END_VAR
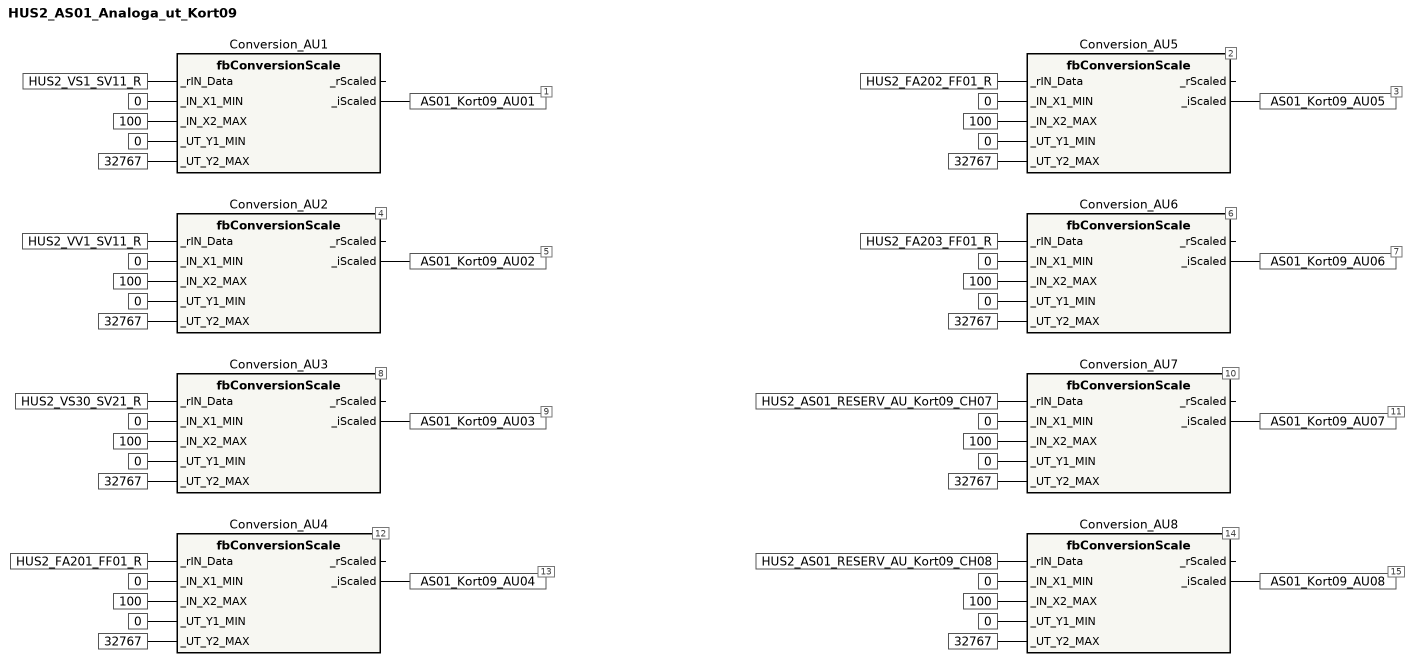
[picture p38: HUS2_AS01_Analoga_ut_Kort09 (CFC)]
_CFC_ (* Continuous Function Chart, elements in execution order *)
#0 Conversion_AU1:fbConversionScale(_rIN_Data: HUS2_VS1_SV11_R, _IN_X1_MIN: 0, _IN_X2_MAX: 100, _UT_Y1_MIN: 0, _UT_Y2_MAX: 32767)
#1 AS01_Kort09_AU01 <= #0._iScaled
#2 Conversion_AU5:fbConversionScale(_rIN_Data: HUS2_FA202_FF01_R, _IN_X1_MIN: 0, _IN_X2_MAX: 100, _UT_Y1_MIN: 0, _UT_Y2_MAX: 32767)
#3 AS01_Kort09_AU05 <= #2._iScaled
#4 Conversion_AU2:fbConversionScale(_rIN_Data: HUS2_VV1_SV11_R, _IN_X1_MIN: 0, _IN_X2_MAX: 100, _UT_Y1_MIN: 0, _UT_Y2_MAX: 32767)
#5 AS01_Kort09_AU02 <= #4._iScaled
#6 Conversion_AU6:fbConversionScale(_rIN_Data: HUS2_FA203_FF01_R, _IN_X1_MIN: 0, _IN_X2_MAX: 100, _UT_Y1_MIN: 0, _UT_Y2_MAX: 32767)
#7 AS01_Kort09_AU06 <= #6._iScaled
#8 Conversion_AU3:fbConversionScale(_rIN_Data: HUS2_VS30_SV21_R, _IN_X1_MIN: 0, _IN_X2_MAX: 100, _UT_Y1_MIN: 0, _UT_Y2_MAX: 32767)
#9 AS01_Kort09_AU03 <= #8._iScaled
#10 Conversion_AU7:fbConversionScale(_rIN_Data: HUS2_AS01_RESERV_AU_Kort09_CH07, _IN_X1_MIN: 0, _IN_X2_MAX: 100, _UT_Y1_MIN: 0, _UT_Y2_MAX: 32767)
#11 AS01_Kort09_AU07 <= #10._iScaled
#12 Conversion_AU4:fbConversionScale(_rIN_Data: HUS2_FA201_FF01_R, _IN_X1_MIN: 0, _IN_X2_MAX: 100, _UT_Y1_MIN: 0, _UT_Y2_MAX: 32767)
#13 AS01_Kort09_AU04 <= #12._iScaled
#14 Conversion_AU8:fbConversionScale(_rIN_Data: HUS2_AS01_RESERV_AU_Kort09_CH08, _IN_X1_MIN: 0, _IN_X2_MAX: 100, _UT_Y1_MIN: 0, _UT_Y2_MAX: 32767)
#15 AS01_Kort09_AU08 <= #14._iScaled
_END_CFC_
(* the same logic as Structured Text *)
Conversion_AU1(_rIN_Data := HUS2_VS1_SV11_R, _IN_X1_MIN := 0, _IN_X2_MAX := 100, _UT_Y1_MIN := 0, _UT_Y2_MAX := 32767);
AS01_Kort09_AU01 := Conversion_AU1._iScaled;
Conversion_AU5(_rIN_Data := HUS2_FA202_FF01_R, _IN_X1_MIN := 0, _IN_X2_MAX := 100, _UT_Y1_MIN := 0, _UT_Y2_MAX := 32767);
AS01_Kort09_AU05 := Conversion_AU5._iScaled;
Conversion_AU2(_rIN_Data := HUS2_VV1_SV11_R, _IN_X1_MIN := 0, _IN_X2_MAX := 100, _UT_Y1_MIN := 0, _UT_Y2_MAX := 32767);
AS01_Kort09_AU02 := Conversion_AU2._iScaled;
Conversion_AU6(_rIN_Data := HUS2_FA203_FF01_R, _IN_X1_MIN := 0, _IN_X2_MAX := 100, _UT_Y1_MIN := 0, _UT_Y2_MAX := 32767);
AS01_Kort09_AU06 := Conversion_AU6._iScaled;
Conversion_AU3(_rIN_Data := HUS2_VS30_SV21_R, _IN_X1_MIN := 0, _IN_X2_MAX := 100, _UT_Y1_MIN := 0, _UT_Y2_MAX := 32767);
AS01_Kort09_AU03 := Conversion_AU3._iScaled;
Conversion_AU7(_rIN_Data := HUS2_AS01_RESERV_AU_Kort09_CH07, _IN_X1_MIN := 0, _IN_X2_MAX := 100, _UT_Y1_MIN := 0, _UT_Y2_MAX := 32767);
AS01_Kort09_AU07 := Conversion_AU7._iScaled;
Conversion_AU4(_rIN_Data := HUS2_FA201_FF01_R, _IN_X1_MIN := 0, _IN_X2_MAX := 100, _UT_Y1_MIN := 0, _UT_Y2_MAX := 32767);
AS01_Kort09_AU04 := Conversion_AU4._iScaled;
Conversion_AU8(_rIN_Data := HUS2_AS01_RESERV_AU_Kort09_CH08, _IN_X1_MIN := 0, _IN_X2_MAX := 100, _UT_Y1_MIN := 0, _UT_Y2_MAX := 32767);
AS01_Kort09_AU08 := Conversion_AU8._iScaled;
END_PROGRAM

(* POU _IOs_Uppdelat_per_skåp/HUS2_AL01/_IO/HUS2_AL01_IO_MAIN, CFC *)
PROGRAM HUS2_AL01_IO_MAIN
VAR
END_VAR
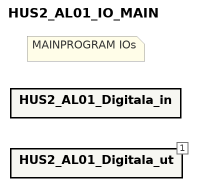
_CFC_ (* Continuous Function Chart, elements in execution order *)
(* MAINPROGRAM IOs *)
#0 HUS2_AL01_Digitala_in()
#1 HUS2_AL01_Digitala_ut()
_END_CFC_
(* the same logic as Structured Text *)
(* MAINPROGRAM IOs *)
HUS2_AL01_Digitala_in();
HUS2_AL01_Digitala_ut();
END_PROGRAM

(* POU _IOs_Uppdelat_per_skåp/HUS2_AL01/_IO/HUS2_AL01_Digitala_in, CFC *)
PROGRAM HUS2_AL01_Digitala_in

VAR


END_VAR
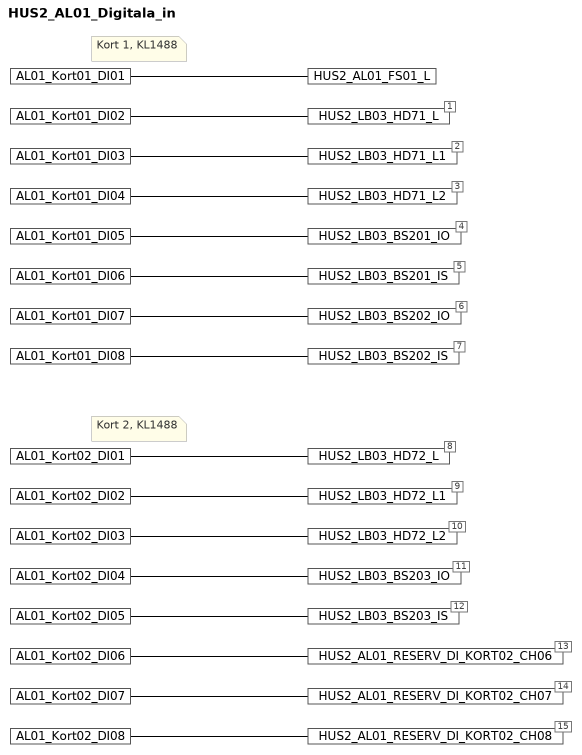
_CFC_ (* Continuous Function Chart, elements in execution order *)
(* Kort 1, KL1488 *)
(* Kort 2, KL1488 *)
#0 HUS2_AL01_FS01_L <= AL01_Kort01_DI01
#1 HUS2_LB03_HD71_L <= AL01_Kort01_DI02
#2 HUS2_LB03_HD71_L1 <= AL01_Kort01_DI03
#3 HUS2_LB03_HD71_L2 <= AL01_Kort01_DI04
#4 HUS2_LB03_BS201_IO <= AL01_Kort01_DI05
#5 HUS2_LB03_BS201_IS <= AL01_Kort01_DI06
#6 HUS2_LB03_BS202_IO <= AL01_Kort01_DI07
#7 HUS2_LB03_BS202_IS <= AL01_Kort01_DI08
#8 HUS2_LB03_HD72_L <= AL01_Kort02_DI01
#9 HUS2_LB03_HD72_L1 <= AL01_Kort02_DI02
#10 HUS2_LB03_HD72_L2 <= AL01_Kort02_DI03
#11 HUS2_LB03_BS203_IO <= AL01_Kort02_DI04
#12 HUS2_LB03_BS203_IS <= AL01_Kort02_DI05
#13 HUS2_AL01_RESERV_DI_KORT02_CH06 <= AL01_Kort02_DI06
#14 HUS2_AL01_RESERV_DI_KORT02_CH07 <= AL01_Kort02_DI07
#15 HUS2_AL01_RESERV_DI_KORT02_CH08 <= AL01_Kort02_DI08
_END_CFC_
(* the same logic as Structured Text *)
(* Kort 1, KL1488 *)
(* Kort 2, KL1488 *)
HUS2_AL01_FS01_L := AL01_Kort01_DI01;
HUS2_LB03_HD71_L := AL01_Kort01_DI02;
HUS2_LB03_HD71_L1 := AL01_Kort01_DI03;
HUS2_LB03_HD71_L2 := AL01_Kort01_DI04;
HUS2_LB03_BS201_IO := AL01_Kort01_DI05;
HUS2_LB03_BS201_IS := AL01_Kort01_DI06;
HUS2_LB03_BS202_IO := AL01_Kort01_DI07;
HUS2_LB03_BS202_IS := AL01_Kort01_DI08;
HUS2_LB03_HD72_L := AL01_Kort02_DI01;
HUS2_LB03_HD72_L1 := AL01_Kort02_DI02;
HUS2_LB03_HD72_L2 := AL01_Kort02_DI03;
HUS2_LB03_BS203_IO := AL01_Kort02_DI04;
HUS2_LB03_BS203_IS := AL01_Kort02_DI05;
HUS2_AL01_RESERV_DI_KORT02_CH06 := AL01_Kort02_DI06;
HUS2_AL01_RESERV_DI_KORT02_CH07 := AL01_Kort02_DI07;
HUS2_AL01_RESERV_DI_KORT02_CH08 := AL01_Kort02_DI08;
END_PROGRAM

(* POU _IOs_Uppdelat_per_skåp/HUS2_AL01/_IO/HUS2_AL01_Digitala_ut, CFC *)
PROGRAM HUS2_AL01_Digitala_ut


VAR
END_VAR
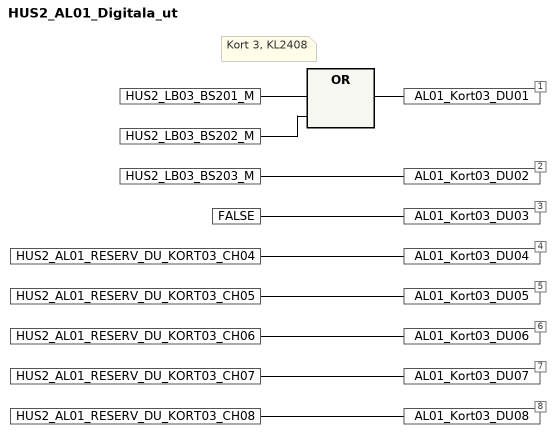
_CFC_ (* Continuous Function Chart, elements in execution order *)
(* Kort 3, KL2408 *)
#0 OR(HUS2_LB03_BS201_M, HUS2_LB03_BS202_M)
#1 AL01_Kort03_DU01 <= #0
#2 AL01_Kort03_DU02 <= HUS2_LB03_BS203_M
#3 AL01_Kort03_DU03 <= FALSE
#4 AL01_Kort03_DU04 <= HUS2_AL01_RESERV_DU_KORT03_CH04
#5 AL01_Kort03_DU05 <= HUS2_AL01_RESERV_DU_KORT03_CH05
#6 AL01_Kort03_DU06 <= HUS2_AL01_RESERV_DU_KORT03_CH06
#7 AL01_Kort03_DU07 <= HUS2_AL01_RESERV_DU_KORT03_CH07
#8 AL01_Kort03_DU08 <= HUS2_AL01_RESERV_DU_KORT03_CH08
_END_CFC_
(* the same logic as Structured Text *)
(* Kort 3, KL2408 *)
AL01_Kort03_DU01 := HUS2_LB03_BS201_M OR HUS2_LB03_BS202_M;
AL01_Kort03_DU02 := HUS2_LB03_BS203_M;
AL01_Kort03_DU03 := FALSE;
AL01_Kort03_DU04 := HUS2_AL01_RESERV_DU_KORT03_CH04;
AL01_Kort03_DU05 := HUS2_AL01_RESERV_DU_KORT03_CH05;
AL01_Kort03_DU06 := HUS2_AL01_RESERV_DU_KORT03_CH06;
AL01_Kort03_DU07 := HUS2_AL01_RESERV_DU_KORT03_CH07;
AL01_Kort03_DU08 := HUS2_AL01_RESERV_DU_KORT03_CH08;
END_PROGRAM

(* POU _IOs_Uppdelat_per_skåp/HUS3_AS03/_IO/HUS3_AS03_IO_MAIN, CFC *)
PROGRAM HUS3_AS03_IO_MAIN
VAR
END_VAR
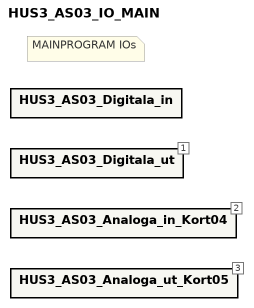
_CFC_ (* Continuous Function Chart, elements in execution order *)
(* MAINPROGRAM IOs *)
#0 HUS3_AS03_Digitala_in()
#1 HUS3_AS03_Digitala_ut()
#2 HUS3_AS03_Analoga_in_Kort04()
#3 HUS3_AS03_Analoga_ut_Kort05()
_END_CFC_
(* the same logic as Structured Text *)
(* MAINPROGRAM IOs *)
HUS3_AS03_Digitala_in();
HUS3_AS03_Digitala_ut();
HUS3_AS03_Analoga_in_Kort04();
HUS3_AS03_Analoga_ut_Kort05();
END_PROGRAM

(* POU _IOs_Uppdelat_per_skåp/HUS3_AS03/_IO/HUS3_AS03_Digitala_in, CFC *)
PROGRAM HUS3_AS03_Digitala_in

VAR


END_VAR
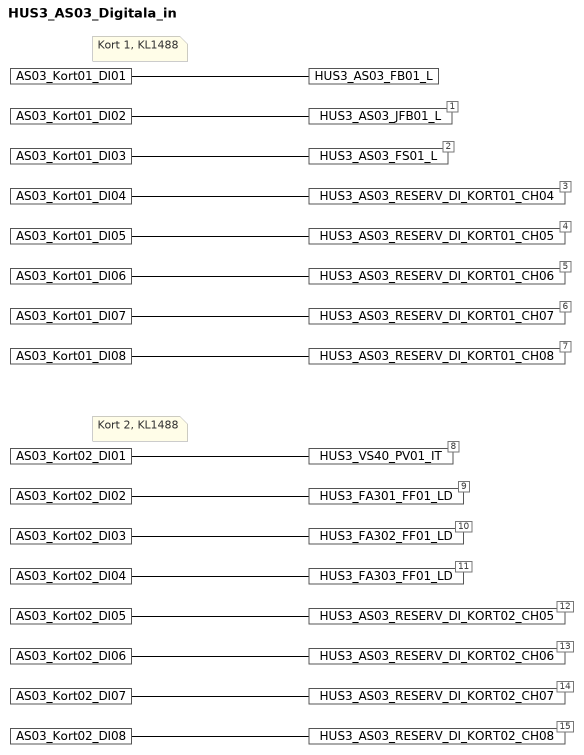
_CFC_ (* Continuous Function Chart, elements in execution order *)
(* Kort 2, KL1488 *)
(* Kort 1, KL1488 *)
#0 HUS3_AS03_FB01_L <= AS03_Kort01_DI01
#1 HUS3_AS03_JFB01_L <= AS03_Kort01_DI02
#2 HUS3_AS03_FS01_L <= AS03_Kort01_DI03
#3 HUS3_AS03_RESERV_DI_KORT01_CH04 <= AS03_Kort01_DI04
#4 HUS3_AS03_RESERV_DI_KORT01_CH05 <= AS03_Kort01_DI05
#5 HUS3_AS03_RESERV_DI_KORT01_CH06 <= AS03_Kort01_DI06
#6 HUS3_AS03_RESERV_DI_KORT01_CH07 <= AS03_Kort01_DI07
#7 HUS3_AS03_RESERV_DI_KORT01_CH08 <= AS03_Kort01_DI08
#8 HUS3_VS40_PV01_IT <= AS03_Kort02_DI01
#9 HUS3_FA301_FF01_LD <= AS03_Kort02_DI02
#10 HUS3_FA302_FF01_LD <= AS03_Kort02_DI03
#11 HUS3_FA303_FF01_LD <= AS03_Kort02_DI04
#12 HUS3_AS03_RESERV_DI_KORT02_CH05 <= AS03_Kort02_DI05
#13 HUS3_AS03_RESERV_DI_KORT02_CH06 <= AS03_Kort02_DI06
#14 HUS3_AS03_RESERV_DI_KORT02_CH07 <= AS03_Kort02_DI07
#15 HUS3_AS03_RESERV_DI_KORT02_CH08 <= AS03_Kort02_DI08
_END_CFC_
(* the same logic as Structured Text *)
(* Kort 2, KL1488 *)
(* Kort 1, KL1488 *)
HUS3_AS03_FB01_L := AS03_Kort01_DI01;
HUS3_AS03_JFB01_L := AS03_Kort01_DI02;
HUS3_AS03_FS01_L := AS03_Kort01_DI03;
HUS3_AS03_RESERV_DI_KORT01_CH04 := AS03_Kort01_DI04;
HUS3_AS03_RESERV_DI_KORT01_CH05 := AS03_Kort01_DI05;
HUS3_AS03_RESERV_DI_KORT01_CH06 := AS03_Kort01_DI06;
HUS3_AS03_RESERV_DI_KORT01_CH07 := AS03_Kort01_DI07;
HUS3_AS03_RESERV_DI_KORT01_CH08 := AS03_Kort01_DI08;
HUS3_VS40_PV01_IT := AS03_Kort02_DI01;
HUS3_FA301_FF01_LD := AS03_Kort02_DI02;
HUS3_FA302_FF01_LD := AS03_Kort02_DI03;
HUS3_FA303_FF01_LD := AS03_Kort02_DI04;
HUS3_AS03_RESERV_DI_KORT02_CH05 := AS03_Kort02_DI05;
HUS3_AS03_RESERV_DI_KORT02_CH06 := AS03_Kort02_DI06;
HUS3_AS03_RESERV_DI_KORT02_CH07 := AS03_Kort02_DI07;
HUS3_AS03_RESERV_DI_KORT02_CH08 := AS03_Kort02_DI08;
END_PROGRAM

(* POU _IOs_Uppdelat_per_skåp/HUS3_AS03/_IO/HUS3_AS03_Digitala_ut, CFC *)
PROGRAM HUS3_AS03_Digitala_ut


VAR

END_VAR
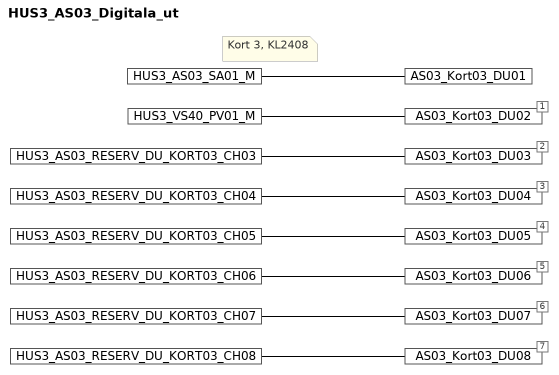
_CFC_ (* Continuous Function Chart, elements in execution order *)
(* Kort 3, KL2408 *)
#0 AS03_Kort03_DU01 <= HUS3_AS03_SA01_M
#1 AS03_Kort03_DU02 <= HUS3_VS40_PV01_M
#2 AS03_Kort03_DU03 <= HUS3_AS03_RESERV_DU_KORT03_CH03
#3 AS03_Kort03_DU04 <= HUS3_AS03_RESERV_DU_KORT03_CH04
#4 AS03_Kort03_DU05 <= HUS3_AS03_RESERV_DU_KORT03_CH05
#5 AS03_Kort03_DU06 <= HUS3_AS03_RESERV_DU_KORT03_CH06
#6 AS03_Kort03_DU07 <= HUS3_AS03_RESERV_DU_KORT03_CH07
#7 AS03_Kort03_DU08 <= HUS3_AS03_RESERV_DU_KORT03_CH08
_END_CFC_
(* the same logic as Structured Text *)
(* Kort 3, KL2408 *)
AS03_Kort03_DU01 := HUS3_AS03_SA01_M;
AS03_Kort03_DU02 := HUS3_VS40_PV01_M;
AS03_Kort03_DU03 := HUS3_AS03_RESERV_DU_KORT03_CH03;
AS03_Kort03_DU04 := HUS3_AS03_RESERV_DU_KORT03_CH04;
AS03_Kort03_DU05 := HUS3_AS03_RESERV_DU_KORT03_CH05;
AS03_Kort03_DU06 := HUS3_AS03_RESERV_DU_KORT03_CH06;
AS03_Kort03_DU07 := HUS3_AS03_RESERV_DU_KORT03_CH07;
AS03_Kort03_DU08 := HUS3_AS03_RESERV_DU_KORT03_CH08;
END_PROGRAM

(* POU _IOs_Uppdelat_per_skåp/HUS3_AS03/_IO/ANALOGA IN/Kort04/HUS3_AS03_Analoga_in_Kort04, CFC *)
PROGRAM HUS3_AS03_Analoga_in_Kort04
VAR
	bLG01: BOOL;
	bLG02: BOOL;
	bLG03: BOOL;
	bLG04: BOOL;
	bLG05: BOOL;
	bLG06: BOOL;
	bLG07: BOOL;
	bLG08: BOOL;

(*TEMP*)
	FT1:INT;
	LG_FL1:INT;
	FT2:INT;
	LG_FL2:INT;
	FT3:INT;
	LG_FL3:INT;
	FT4:INT;
	LG_FL4:INT;
	FT5:INT;
	LG_FL5:INT;
	FT6:INT;
	LG_FL6:INT;
	FT7:INT;
	LG_FL7:INT;
	FT8:INT;
	LG_FL8:INT;

END_VAR
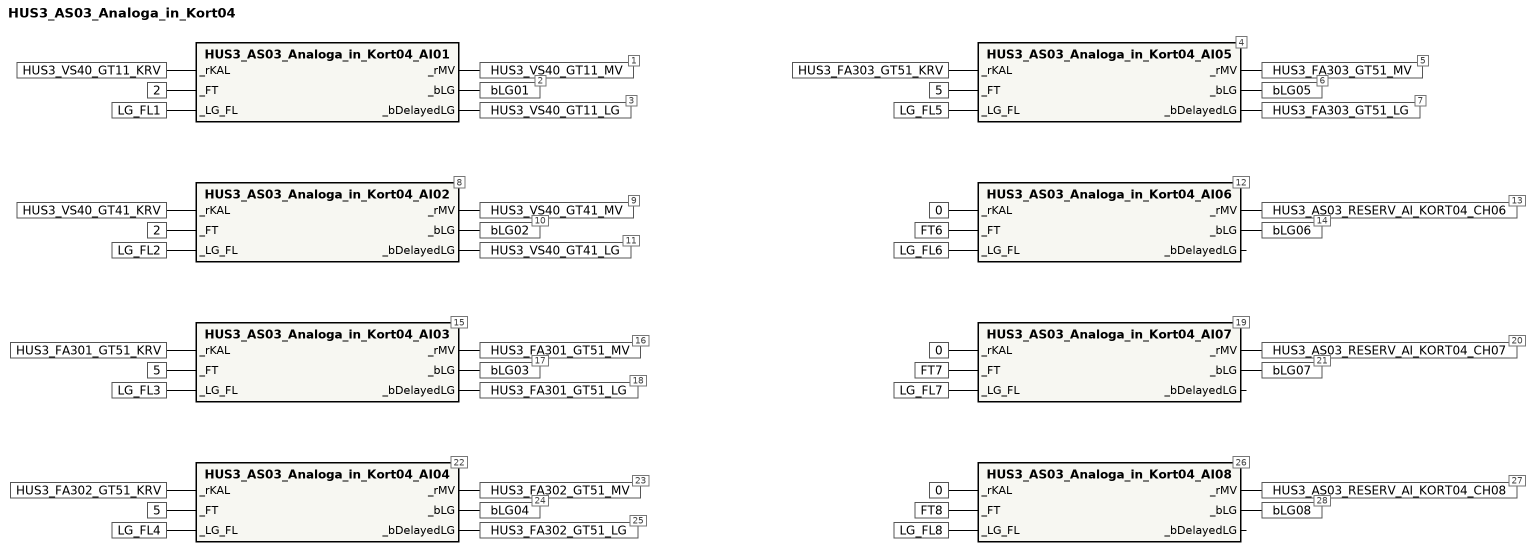
_CFC_ (* Continuous Function Chart, elements in execution order *)
#0 HUS3_AS03_Analoga_in_Kort04_AI01(_rKAL: HUS3_VS40_GT11_KRV, _FT: 2, _LG_FL: LG_FL1)
#1 HUS3_VS40_GT11_MV <= #0._rMV
#2 bLG01 <= #0._bLG
#3 HUS3_VS40_GT11_LG <= #0._bDelayedLG
#4 HUS3_AS03_Analoga_in_Kort04_AI05(_rKAL: HUS3_FA303_GT51_KRV, _FT: 5, _LG_FL: LG_FL5)
#5 HUS3_FA303_GT51_MV <= #4._rMV
#6 bLG05 <= #4._bLG
#7 HUS3_FA303_GT51_LG <= #4._bDelayedLG
#8 HUS3_AS03_Analoga_in_Kort04_AI02(_rKAL: HUS3_VS40_GT41_KRV, _FT: 2, _LG_FL: LG_FL2)
#9 HUS3_VS40_GT41_MV <= #8._rMV
#10 bLG02 <= #8._bLG
#11 HUS3_VS40_GT41_LG <= #8._bDelayedLG
#12 HUS3_AS03_Analoga_in_Kort04_AI06(_rKAL: 0, _FT: FT6, _LG_FL: LG_FL6)
#13 HUS3_AS03_RESERV_AI_KORT04_CH06 <= #12._rMV
#14 bLG06 <= #12._bLG
#15 HUS3_AS03_Analoga_in_Kort04_AI03(_rKAL: HUS3_FA301_GT51_KRV, _FT: 5, _LG_FL: LG_FL3)
#16 HUS3_FA301_GT51_MV <= #15._rMV
#17 bLG03 <= #15._bLG
#18 HUS3_FA301_GT51_LG <= #15._bDelayedLG
#19 HUS3_AS03_Analoga_in_Kort04_AI07(_rKAL: 0, _FT: FT7, _LG_FL: LG_FL7)
#20 HUS3_AS03_RESERV_AI_KORT04_CH07 <= #19._rMV
#21 bLG07 <= #19._bLG
#22 HUS3_AS03_Analoga_in_Kort04_AI04(_rKAL: HUS3_FA302_GT51_KRV, _FT: 5, _LG_FL: LG_FL4)
#23 HUS3_FA302_GT51_MV <= #22._rMV
#24 bLG04 <= #22._bLG
#25 HUS3_FA302_GT51_LG <= #22._bDelayedLG
#26 HUS3_AS03_Analoga_in_Kort04_AI08(_rKAL: 0, _FT: FT8, _LG_FL: LG_FL8)
#27 HUS3_AS03_RESERV_AI_KORT04_CH08 <= #26._rMV
#28 bLG08 <= #26._bLG
_END_CFC_
(* the same logic as Structured Text *)
HUS3_AS03_Analoga_in_Kort04_AI01(_rKAL := HUS3_VS40_GT11_KRV, _FT := 2, _LG_FL := LG_FL1);
HUS3_VS40_GT11_MV := HUS3_AS03_Analoga_in_Kort04_AI01._rMV;
bLG01 := HUS3_AS03_Analoga_in_Kort04_AI01._bLG;
HUS3_VS40_GT11_LG := HUS3_AS03_Analoga_in_Kort04_AI01._bDelayedLG;
HUS3_AS03_Analoga_in_Kort04_AI05(_rKAL := HUS3_FA303_GT51_KRV, _FT := 5, _LG_FL := LG_FL5);
HUS3_FA303_GT51_MV := HUS3_AS03_Analoga_in_Kort04_AI05._rMV;
bLG05 := HUS3_AS03_Analoga_in_Kort04_AI05._bLG;
HUS3_FA303_GT51_LG := HUS3_AS03_Analoga_in_Kort04_AI05._bDelayedLG;
HUS3_AS03_Analoga_in_Kort04_AI02(_rKAL := HUS3_VS40_GT41_KRV, _FT := 2, _LG_FL := LG_FL2);
HUS3_VS40_GT41_MV := HUS3_AS03_Analoga_in_Kort04_AI02._rMV;
bLG02 := HUS3_AS03_Analoga_in_Kort04_AI02._bLG;
HUS3_VS40_GT41_LG := HUS3_AS03_Analoga_in_Kort04_AI02._bDelayedLG;
HUS3_AS03_Analoga_in_Kort04_AI06(_rKAL := 0, _FT := FT6, _LG_FL := LG_FL6);
HUS3_AS03_RESERV_AI_KORT04_CH06 := HUS3_AS03_Analoga_in_Kort04_AI06._rMV;
bLG06 := HUS3_AS03_Analoga_in_Kort04_AI06._bLG;
HUS3_AS03_Analoga_in_Kort04_AI03(_rKAL := HUS3_FA301_GT51_KRV, _FT := 5, _LG_FL := LG_FL3);
HUS3_FA301_GT51_MV := HUS3_AS03_Analoga_in_Kort04_AI03._rMV;
bLG03 := HUS3_AS03_Analoga_in_Kort04_AI03._bLG;
HUS3_FA301_GT51_LG := HUS3_AS03_Analoga_in_Kort04_AI03._bDelayedLG;
HUS3_AS03_Analoga_in_Kort04_AI07(_rKAL := 0, _FT := FT7, _LG_FL := LG_FL7);
HUS3_AS03_RESERV_AI_KORT04_CH07 := HUS3_AS03_Analoga_in_Kort04_AI07._rMV;
bLG07 := HUS3_AS03_Analoga_in_Kort04_AI07._bLG;
HUS3_AS03_Analoga_in_Kort04_AI04(_rKAL := HUS3_FA302_GT51_KRV, _FT := 5, _LG_FL := LG_FL4);
HUS3_FA302_GT51_MV := HUS3_AS03_Analoga_in_Kort04_AI04._rMV;
bLG04 := HUS3_AS03_Analoga_in_Kort04_AI04._bLG;
HUS3_FA302_GT51_LG := HUS3_AS03_Analoga_in_Kort04_AI04._bDelayedLG;
HUS3_AS03_Analoga_in_Kort04_AI08(_rKAL := 0, _FT := FT8, _LG_FL := LG_FL8);
HUS3_AS03_RESERV_AI_KORT04_CH08 := HUS3_AS03_Analoga_in_Kort04_AI08._rMV;
bLG08 := HUS3_AS03_Analoga_in_Kort04_AI08._bLG;
END_PROGRAM

(* POU _IOs_Uppdelat_per_skåp/HUS3_AS03/_IO/ANALOGA IN/Kort04/HUS3_AS03_Analoga_in_Kort04_AI01, FAI *)
PROGRAM HUS3_AS03_Analoga_in_Kort04_AI01
(*#####################################   Temperature Sensor Ex2   ################################################################*)
VAR
	(*===========================Configuration of terminal==========================================*)
	fbConfigureKL32xx					:FB_HVACConfigureKL32xx;
	_byCtrlKL32xx                         			AT %Q*: BYTE;
	_iDataOutKL32xx                       		AT %Q*: INT;
	_iDataInKL32xx 					AT%I*:INT;(* Raw Value from the Terminal *)
	_byStatusKL32xx 			AT%I*:BYTE;(* Statusbyte from Terminal *)

	_bScanSensor              					: BOOL;
	_tTimeOut                 					: TIME := T#5s;
	_bSetSensor               					: BOOL;
	bReady                               				: BOOL;
	byOutStatus                          			: BYTE;
	iOutDataIn                           				: INT;
	_eBusTerminalKL32xx                   		: E_HVACBusTerminal_KL32xx;
	_eStatusScanSensorType                	: E_HVACSensorType;
	_bErrorGeneral                        			: BOOL;
	_byError                              				: BYTE;
	_bErrorCommunication                  		: BOOL;
	_bErrorBusTerminalNotSupported   	: BOOL;
	_bErrorSensorType                     		: BOOL;
	_bErrorScanSensor                     		: BOOL;
	(*========================================================================================*)

	_bReset_Local					:BOOL;
	_bSetDefaultTempSens			:BOOL;

	(*========================================================================================*)
	FBHVACTemperatureSensor: FB_HVACTemperatureSensor;
	eDataSecurityType					: E_HVACDataSecurityType:=1;
	bSetDefault								:BOOL;
	iRawValue								:INT;
	byStatusRawValue						:BYTE;
	bEnableLimitCtrl							:BOOL;
	bReset									:BOOL;
	bErrorGeneral					:BOOL;
	byError							:BYTE;
	bErrorShortCircuit				:BOOL;
	bErrorBrokenSensor				:BOOL;
	bErrorHighLimit					:BOOL;
	bErrorLowLimit					:BOOL;
	bErrorCycleTime					:BOOL;
	bInvalidParameter				:BOOL;
	rOffset									:REAL;
	rHighLimit								:REAL;
	rLowLimit								:REAL;
	rReplacementValue						:REAL;
	tFilterTime								:TIME;
	eTemperatureSensorMode				:E_HVACTemperatureSensorMode:=2;
	fbAlarmD: fbDelayedAlarmMinutes;

END_VAR

VAR_INPUT
	_rKAL						: REAL;	(*Kalibrering*)
	_FT						:INT;		(*Filtertid*)
	_LG_FL					:INT;		(* Larmfördröjning givarfel *)
END_VAR

VAR_OUTPUT
	_rMV						:REAL;		(* Mätvärde *)
	_bLG						:BOOL; 	(*Givarfel*)
	_bDelayedLG				:BOOL;	(* Fördröjt givarfel *)
END_VAR
(* body not read: cfc101 *)
END_PROGRAM

(* POU _IOs_Uppdelat_per_skåp/HUS3_AS03/_IO/ANALOGA IN/Kort04/HUS3_AS03_Analoga_in_Kort04_AI05, FAI *)
PROGRAM HUS3_AS03_Analoga_in_Kort04_AI05
(*#####################################   Temperature Sensor Ex2   ################################################################*)
VAR
	(*===========================Configuration of terminal==========================================*)
	fbConfigureKL32xx					:FB_HVACConfigureKL32xx;
	_byCtrlKL32xx                         			AT %Q*: BYTE;
	_iDataOutKL32xx                       		AT %Q*: INT;
	_iDataInKL32xx 					AT%I*:INT;(* Raw Value from the Terminal *)
	_byStatusKL32xx 			AT%I*:BYTE;(* Statusbyte from Terminal *)

	_bScanSensor              					: BOOL;
	_tTimeOut                 					: TIME := T#5s;
	_bSetSensor               					: BOOL;
	bReady                               				: BOOL;
	byOutStatus                          			: BYTE;
	iOutDataIn                           				: INT;
	_eBusTerminalKL32xx                   		: E_HVACBusTerminal_KL32xx;
	_eStatusScanSensorType                	: E_HVACSensorType;
	_bErrorGeneral                        			: BOOL;
	_byError                              				: BYTE;
	_bErrorCommunication                  		: BOOL;
	_bErrorBusTerminalNotSupported   	: BOOL;
	_bErrorSensorType                     		: BOOL;
	_bErrorScanSensor                     		: BOOL;
	(*========================================================================================*)

	_bReset_Local					:BOOL;
	_bSetDefaultTempSens			:BOOL;

	(*========================================================================================*)
	FBHVACTemperatureSensor: FB_HVACTemperatureSensor;
	eDataSecurityType					: E_HVACDataSecurityType:=1;
	bSetDefault								:BOOL;
	iRawValue								:INT;
	byStatusRawValue						:BYTE;
	bEnableLimitCtrl							:BOOL;
	bReset									:BOOL;
	bErrorGeneral					:BOOL;
	byError							:BYTE;
	bErrorShortCircuit				:BOOL;
	bErrorBrokenSensor				:BOOL;
	bErrorHighLimit					:BOOL;
	bErrorLowLimit					:BOOL;
	bErrorCycleTime					:BOOL;
	bInvalidParameter				:BOOL;
	rOffset									:REAL;
	rHighLimit								:REAL;
	rLowLimit								:REAL;
	rReplacementValue						:REAL;
	tFilterTime								:TIME;
	eTemperatureSensorMode				:E_HVACTemperatureSensorMode:=2;
	fbAlarmD: fbDelayedAlarmMinutes;

END_VAR

VAR_INPUT
	_rKAL						: REAL;	(*Kalibrering*)
	_FT						:INT;		(*Filtertid*)
	_LG_FL					:INT;		(* Larmfördröjning givarfel *)
END_VAR

VAR_OUTPUT
	_rMV						:REAL;		(* Mätvärde *)
	_bLG						:BOOL; 	(*Givarfel*)
	_bDelayedLG				:BOOL;	(* Fördröjt givarfel *)
END_VAR
(* body not read: cfc101 *)
END_PROGRAM

(* POU _IOs_Uppdelat_per_skåp/HUS3_AS03/_IO/ANALOGA IN/Kort04/HUS3_AS03_Analoga_in_Kort04_AI02, FAI *)
PROGRAM HUS3_AS03_Analoga_in_Kort04_AI02
(*#####################################   Temperature Sensor Ex2   ################################################################*)
VAR
	(*===========================Configuration of terminal==========================================*)
	fbConfigureKL32xx					:FB_HVACConfigureKL32xx;
	_byCtrlKL32xx                         			AT %Q*: BYTE;
	_iDataOutKL32xx                       		AT %Q*: INT;
	_iDataInKL32xx 					AT%I*:INT;(* Raw Value from the Terminal *)
	_byStatusKL32xx 			AT%I*:BYTE;(* Statusbyte from Terminal *)

	_bScanSensor              					: BOOL;
	_tTimeOut                 					: TIME := T#5s;
	_bSetSensor               					: BOOL;
	bReady                               				: BOOL;
	byOutStatus                          			: BYTE;
	iOutDataIn                           				: INT;
	_eBusTerminalKL32xx                   		: E_HVACBusTerminal_KL32xx;
	_eStatusScanSensorType                	: E_HVACSensorType;
	_bErrorGeneral                        			: BOOL;
	_byError                              				: BYTE;
	_bErrorCommunication                  		: BOOL;
	_bErrorBusTerminalNotSupported   	: BOOL;
	_bErrorSensorType                     		: BOOL;
	_bErrorScanSensor                     		: BOOL;
	(*========================================================================================*)

	_bReset_Local					:BOOL;
	_bSetDefaultTempSens			:BOOL;

	(*========================================================================================*)
	FBHVACTemperatureSensor: FB_HVACTemperatureSensor;
	eDataSecurityType					: E_HVACDataSecurityType:=1;
	bSetDefault								:BOOL;
	iRawValue								:INT;
	byStatusRawValue						:BYTE;
	bEnableLimitCtrl							:BOOL;
	bReset									:BOOL;
	bErrorGeneral					:BOOL;
	byError							:BYTE;
	bErrorShortCircuit				:BOOL;
	bErrorBrokenSensor				:BOOL;
	bErrorHighLimit					:BOOL;
	bErrorLowLimit					:BOOL;
	bErrorCycleTime					:BOOL;
	bInvalidParameter				:BOOL;
	rOffset									:REAL;
	rHighLimit								:REAL;
	rLowLimit								:REAL;
	rReplacementValue						:REAL;
	tFilterTime								:TIME;
	eTemperatureSensorMode				:E_HVACTemperatureSensorMode:=2;
	fbAlarmD: fbDelayedAlarmMinutes;

END_VAR

VAR_INPUT
	_rKAL						: REAL;	(*Kalibrering*)
	_FT						:INT;		(*Filtertid*)
	_LG_FL					:INT;		(* Larmfördröjning givarfel *)
END_VAR

VAR_OUTPUT
	_rMV						:REAL;		(* Mätvärde *)
	_bLG						:BOOL; 	(*Givarfel*)
	_bDelayedLG				:BOOL;	(* Fördröjt givarfel *)
END_VAR
(* body not read: cfc101 *)
END_PROGRAM

(* POU _IOs_Uppdelat_per_skåp/HUS3_AS03/_IO/ANALOGA IN/Kort04/HUS3_AS03_Analoga_in_Kort04_AI06, FAI *)
PROGRAM HUS3_AS03_Analoga_in_Kort04_AI06
(*#####################################   Temperature Sensor Ex2   ################################################################*)
VAR
	(*===========================Configuration of terminal==========================================*)
	fbConfigureKL32xx					:FB_HVACConfigureKL32xx;
	_byCtrlKL32xx                         			AT %Q*: BYTE;
	_iDataOutKL32xx                       		AT %Q*: INT;
	_iDataInKL32xx 					AT%I*:INT;(* Raw Value from the Terminal *)
	_byStatusKL32xx 			AT%I*:BYTE;(* Statusbyte from Terminal *)

	_bScanSensor              					: BOOL;
	_tTimeOut                 					: TIME := T#5s;
	_bSetSensor               					: BOOL;
	bReady                               				: BOOL;
	byOutStatus                          			: BYTE;
	iOutDataIn                           				: INT;
	_eBusTerminalKL32xx                   		: E_HVACBusTerminal_KL32xx;
	_eStatusScanSensorType                	: E_HVACSensorType;
	_bErrorGeneral                        			: BOOL;
	_byError                              				: BYTE;
	_bErrorCommunication                  		: BOOL;
	_bErrorBusTerminalNotSupported   	: BOOL;
	_bErrorSensorType                     		: BOOL;
	_bErrorScanSensor                     		: BOOL;
	(*========================================================================================*)

	_bReset_Local					:BOOL;
	_bSetDefaultTempSens			:BOOL;

	(*========================================================================================*)
	FBHVACTemperatureSensor: FB_HVACTemperatureSensor;
	eDataSecurityType					: E_HVACDataSecurityType:=1;
	bSetDefault								:BOOL;
	iRawValue								:INT;
	byStatusRawValue						:BYTE;
	bEnableLimitCtrl							:BOOL;
	bReset									:BOOL;
	bErrorGeneral					:BOOL;
	byError							:BYTE;
	bErrorShortCircuit				:BOOL;
	bErrorBrokenSensor				:BOOL;
	bErrorHighLimit					:BOOL;
	bErrorLowLimit					:BOOL;
	bErrorCycleTime					:BOOL;
	bInvalidParameter				:BOOL;
	rOffset									:REAL;
	rHighLimit								:REAL;
	rLowLimit								:REAL;
	rReplacementValue						:REAL;
	tFilterTime								:TIME;
	eTemperatureSensorMode				:E_HVACTemperatureSensorMode:=2;
	fbAlarmD: fbDelayedAlarmMinutes;

END_VAR

VAR_INPUT
	_rKAL						: REAL;	(*Kalibrering*)
	_FT						:INT;		(*Filtertid*)
	_LG_FL					:INT;		(* Larmfördröjning givarfel *)
END_VAR

VAR_OUTPUT
	_rMV						:REAL;		(* Mätvärde *)
	_bLG						:BOOL; 	(*Givarfel*)
	_bDelayedLG				:BOOL;	(* Fördröjt givarfel *)
END_VAR
(* body not read: cfc101 *)
END_PROGRAM

(* POU _IOs_Uppdelat_per_skåp/HUS3_AS03/_IO/ANALOGA IN/Kort04/HUS3_AS03_Analoga_in_Kort04_AI03, FAI *)
PROGRAM HUS3_AS03_Analoga_in_Kort04_AI03
(*#####################################   Temperature Sensor Ex2   ################################################################*)
VAR
	(*===========================Configuration of terminal==========================================*)
	fbConfigureKL32xx					:FB_HVACConfigureKL32xx;
	_byCtrlKL32xx                         			AT %Q*: BYTE;
	_iDataOutKL32xx                       		AT %Q*: INT;
	_iDataInKL32xx 					AT%I*:INT;(* Raw Value from the Terminal *)
	_byStatusKL32xx 			AT%I*:BYTE;(* Statusbyte from Terminal *)

	_bScanSensor              					: BOOL;
	_tTimeOut                 					: TIME := T#5s;
	_bSetSensor               					: BOOL;
	bReady                               				: BOOL;
	byOutStatus                          			: BYTE;
	iOutDataIn                           				: INT;
	_eBusTerminalKL32xx                   		: E_HVACBusTerminal_KL32xx;
	_eStatusScanSensorType                	: E_HVACSensorType;
	_bErrorGeneral                        			: BOOL;
	_byError                              				: BYTE;
	_bErrorCommunication                  		: BOOL;
	_bErrorBusTerminalNotSupported   	: BOOL;
	_bErrorSensorType                     		: BOOL;
	_bErrorScanSensor                     		: BOOL;
	(*========================================================================================*)

	_bReset_Local					:BOOL;
	_bSetDefaultTempSens			:BOOL;

	(*========================================================================================*)
	FBHVACTemperatureSensor: FB_HVACTemperatureSensor;
	eDataSecurityType					: E_HVACDataSecurityType:=1;
	bSetDefault								:BOOL;
	iRawValue								:INT;
	byStatusRawValue						:BYTE;
	bEnableLimitCtrl							:BOOL;
	bReset									:BOOL;
	bErrorGeneral					:BOOL;
	byError							:BYTE;
	bErrorShortCircuit				:BOOL;
	bErrorBrokenSensor				:BOOL;
	bErrorHighLimit					:BOOL;
	bErrorLowLimit					:BOOL;
	bErrorCycleTime					:BOOL;
	bInvalidParameter				:BOOL;
	rOffset									:REAL;
	rHighLimit								:REAL;
	rLowLimit								:REAL;
	rReplacementValue						:REAL;
	tFilterTime								:TIME;
	eTemperatureSensorMode				:E_HVACTemperatureSensorMode:=2;
	fbAlarmD: fbDelayedAlarmMinutes;

END_VAR

VAR_INPUT
	_rKAL						: REAL;	(*Kalibrering*)
	_FT						:INT;		(*Filtertid*)
	_LG_FL					:INT;		(* Larmfördröjning givarfel *)
END_VAR

VAR_OUTPUT
	_rMV						:REAL;		(* Mätvärde *)
	_bLG						:BOOL; 	(*Givarfel*)
	_bDelayedLG				:BOOL;	(* Fördröjt givarfel *)
END_VAR
(* body not read: cfc101 *)
END_PROGRAM

(* POU _IOs_Uppdelat_per_skåp/HUS3_AS03/_IO/ANALOGA IN/Kort04/HUS3_AS03_Analoga_in_Kort04_AI07, FAI *)
PROGRAM HUS3_AS03_Analoga_in_Kort04_AI07
(*#####################################   Temperature Sensor Ex2   ################################################################*)
VAR
	(*===========================Configuration of terminal==========================================*)
	fbConfigureKL32xx					:FB_HVACConfigureKL32xx;
	_byCtrlKL32xx                         			AT %Q*: BYTE;
	_iDataOutKL32xx                       		AT %Q*: INT;
	_iDataInKL32xx 					AT%I*:INT;(* Raw Value from the Terminal *)
	_byStatusKL32xx 			AT%I*:BYTE;(* Statusbyte from Terminal *)

	_bScanSensor              					: BOOL;
	_tTimeOut                 					: TIME := T#5s;
	_bSetSensor               					: BOOL;
	bReady                               				: BOOL;
	byOutStatus                          			: BYTE;
	iOutDataIn                           				: INT;
	_eBusTerminalKL32xx                   		: E_HVACBusTerminal_KL32xx;
	_eStatusScanSensorType                	: E_HVACSensorType;
	_bErrorGeneral                        			: BOOL;
	_byError                              				: BYTE;
	_bErrorCommunication                  		: BOOL;
	_bErrorBusTerminalNotSupported   	: BOOL;
	_bErrorSensorType                     		: BOOL;
	_bErrorScanSensor                     		: BOOL;
	(*========================================================================================*)

	_bReset_Local					:BOOL;
	_bSetDefaultTempSens			:BOOL;

	(*========================================================================================*)
	FBHVACTemperatureSensor: FB_HVACTemperatureSensor;
	eDataSecurityType					: E_HVACDataSecurityType:=1;
	bSetDefault								:BOOL;
	iRawValue								:INT;
	byStatusRawValue						:BYTE;
	bEnableLimitCtrl							:BOOL;
	bReset									:BOOL;
	bErrorGeneral					:BOOL;
	byError							:BYTE;
	bErrorShortCircuit				:BOOL;
	bErrorBrokenSensor				:BOOL;
	bErrorHighLimit					:BOOL;
	bErrorLowLimit					:BOOL;
	bErrorCycleTime					:BOOL;
	bInvalidParameter				:BOOL;
	rOffset									:REAL;
	rHighLimit								:REAL;
	rLowLimit								:REAL;
	rReplacementValue						:REAL;
	tFilterTime								:TIME;
	eTemperatureSensorMode				:E_HVACTemperatureSensorMode:=2;
	fbAlarmD: fbDelayedAlarmMinutes;

END_VAR

VAR_INPUT
	_rKAL						: REAL;	(*Kalibrering*)
	_FT						:INT;		(*Filtertid*)
	_LG_FL					:INT;		(* Larmfördröjning givarfel *)
END_VAR

VAR_OUTPUT
	_rMV						:REAL;		(* Mätvärde *)
	_bLG						:BOOL; 	(*Givarfel*)
	_bDelayedLG				:BOOL;	(* Fördröjt givarfel *)
END_VAR
(* body not read: cfc101 *)
END_PROGRAM

(* POU _IOs_Uppdelat_per_skåp/HUS3_AS03/_IO/ANALOGA IN/Kort04/HUS3_AS03_Analoga_in_Kort04_AI04, FAI *)
PROGRAM HUS3_AS03_Analoga_in_Kort04_AI04
(*#####################################   Temperature Sensor Ex2   ################################################################*)
VAR
	(*===========================Configuration of terminal==========================================*)
	fbConfigureKL32xx					:FB_HVACConfigureKL32xx;
	_byCtrlKL32xx                         			AT %Q*: BYTE;
	_iDataOutKL32xx                       		AT %Q*: INT;
	_iDataInKL32xx 					AT%I*:INT;(* Raw Value from the Terminal *)
	_byStatusKL32xx 			AT%I*:BYTE;(* Statusbyte from Terminal *)

	_bScanSensor              					: BOOL;
	_tTimeOut                 					: TIME := T#5s;
	_bSetSensor               					: BOOL;
	bReady                               				: BOOL;
	byOutStatus                          			: BYTE;
	iOutDataIn                           				: INT;
	_eBusTerminalKL32xx                   		: E_HVACBusTerminal_KL32xx;
	_eStatusScanSensorType                	: E_HVACSensorType;
	_bErrorGeneral                        			: BOOL;
	_byError                              				: BYTE;
	_bErrorCommunication                  		: BOOL;
	_bErrorBusTerminalNotSupported   	: BOOL;
	_bErrorSensorType                     		: BOOL;
	_bErrorScanSensor                     		: BOOL;
	(*========================================================================================*)

	_bReset_Local					:BOOL;
	_bSetDefaultTempSens			:BOOL;

	(*========================================================================================*)
	FBHVACTemperatureSensor: FB_HVACTemperatureSensor;
	eDataSecurityType					: E_HVACDataSecurityType:=1;
	bSetDefault								:BOOL;
	iRawValue								:INT;
	byStatusRawValue						:BYTE;
	bEnableLimitCtrl							:BOOL;
	bReset									:BOOL;
	bErrorGeneral					:BOOL;
	byError							:BYTE;
	bErrorShortCircuit				:BOOL;
	bErrorBrokenSensor				:BOOL;
	bErrorHighLimit					:BOOL;
	bErrorLowLimit					:BOOL;
	bErrorCycleTime					:BOOL;
	bInvalidParameter				:BOOL;
	rOffset									:REAL;
	rHighLimit								:REAL;
	rLowLimit								:REAL;
	rReplacementValue						:REAL;
	tFilterTime								:TIME;
	eTemperatureSensorMode				:E_HVACTemperatureSensorMode:=2;
	fbAlarmD: fbDelayedAlarmMinutes;

END_VAR

VAR_INPUT
	_rKAL						: REAL;	(*Kalibrering*)
	_FT						:INT;		(*Filtertid*)
	_LG_FL					:INT;		(* Larmfördröjning givarfel *)
END_VAR

VAR_OUTPUT
	_rMV						:REAL;		(* Mätvärde *)
	_bLG						:BOOL; 	(*Givarfel*)
	_bDelayedLG				:BOOL;	(* Fördröjt givarfel *)
END_VAR
(* body not read: cfc101 *)
END_PROGRAM

(* POU _IOs_Uppdelat_per_skåp/HUS3_AS03/_IO/ANALOGA IN/Kort04/HUS3_AS03_Analoga_in_Kort04_AI08, FAI *)
PROGRAM HUS3_AS03_Analoga_in_Kort04_AI08
(*#####################################   Temperature Sensor Ex2   ################################################################*)
VAR
	(*===========================Configuration of terminal==========================================*)
	fbConfigureKL32xx					:FB_HVACConfigureKL32xx;
	_byCtrlKL32xx                         			AT %Q*: BYTE;
	_iDataOutKL32xx                       		AT %Q*: INT;
	_iDataInKL32xx 					AT%I*:INT;(* Raw Value from the Terminal *)
	_byStatusKL32xx 			AT%I*:BYTE;(* Statusbyte from Terminal *)

	_bScanSensor              					: BOOL;
	_tTimeOut                 					: TIME := T#5s;
	_bSetSensor               					: BOOL;
	bReady                               				: BOOL;
	byOutStatus                          			: BYTE;
	iOutDataIn                           				: INT;
	_eBusTerminalKL32xx                   		: E_HVACBusTerminal_KL32xx;
	_eStatusScanSensorType                	: E_HVACSensorType;
	_bErrorGeneral                        			: BOOL;
	_byError                              				: BYTE;
	_bErrorCommunication                  		: BOOL;
	_bErrorBusTerminalNotSupported   	: BOOL;
	_bErrorSensorType                     		: BOOL;
	_bErrorScanSensor                     		: BOOL;
	(*========================================================================================*)

	_bReset_Local					:BOOL;
	_bSetDefaultTempSens			:BOOL;

	(*========================================================================================*)
	FBHVACTemperatureSensor: FB_HVACTemperatureSensor;
	eDataSecurityType					: E_HVACDataSecurityType:=1;
	bSetDefault								:BOOL;
	iRawValue								:INT;
	byStatusRawValue						:BYTE;
	bEnableLimitCtrl							:BOOL;
	bReset									:BOOL;
	bErrorGeneral					:BOOL;
	byError							:BYTE;
	bErrorShortCircuit				:BOOL;
	bErrorBrokenSensor				:BOOL;
	bErrorHighLimit					:BOOL;
	bErrorLowLimit					:BOOL;
	bErrorCycleTime					:BOOL;
	bInvalidParameter				:BOOL;
	rOffset									:REAL;
	rHighLimit								:REAL;
	rLowLimit								:REAL;
	rReplacementValue						:REAL;
	tFilterTime								:TIME;
	eTemperatureSensorMode				:E_HVACTemperatureSensorMode:=2;
	fbAlarmD: fbDelayedAlarmMinutes;

END_VAR

VAR_INPUT
	_rKAL						: REAL;	(*Kalibrering*)
	_FT						:INT;		(*Filtertid*)
	_LG_FL					:INT;		(* Larmfördröjning givarfel *)
END_VAR

VAR_OUTPUT
	_rMV						:REAL;		(* Mätvärde *)
	_bLG						:BOOL; 	(*Givarfel*)
	_bDelayedLG				:BOOL;	(* Fördröjt givarfel *)
END_VAR
(* body not read: cfc101 *)
END_PROGRAM

(* POU _IOs_Uppdelat_per_skåp/HUS3_AS03/_IO/ANALOGA UT/Kort05/HUS3_AS03_Analoga_ut_Kort05, CFC *)
PROGRAM HUS3_AS03_Analoga_ut_Kort05
VAR

	Conversion_AU1: fbConversionScale;
	Conversion_AU2: fbConversionScale;
	Conversion_AU3: fbConversionScale;
	Conversion_AU4: fbConversionScale;
	Conversion_AU5: fbConversionScale;
	Conversion_AU6: fbConversionScale;
	Conversion_AU7: fbConversionScale;
	Conversion_AU8: fbConversionScale;

END_VAR
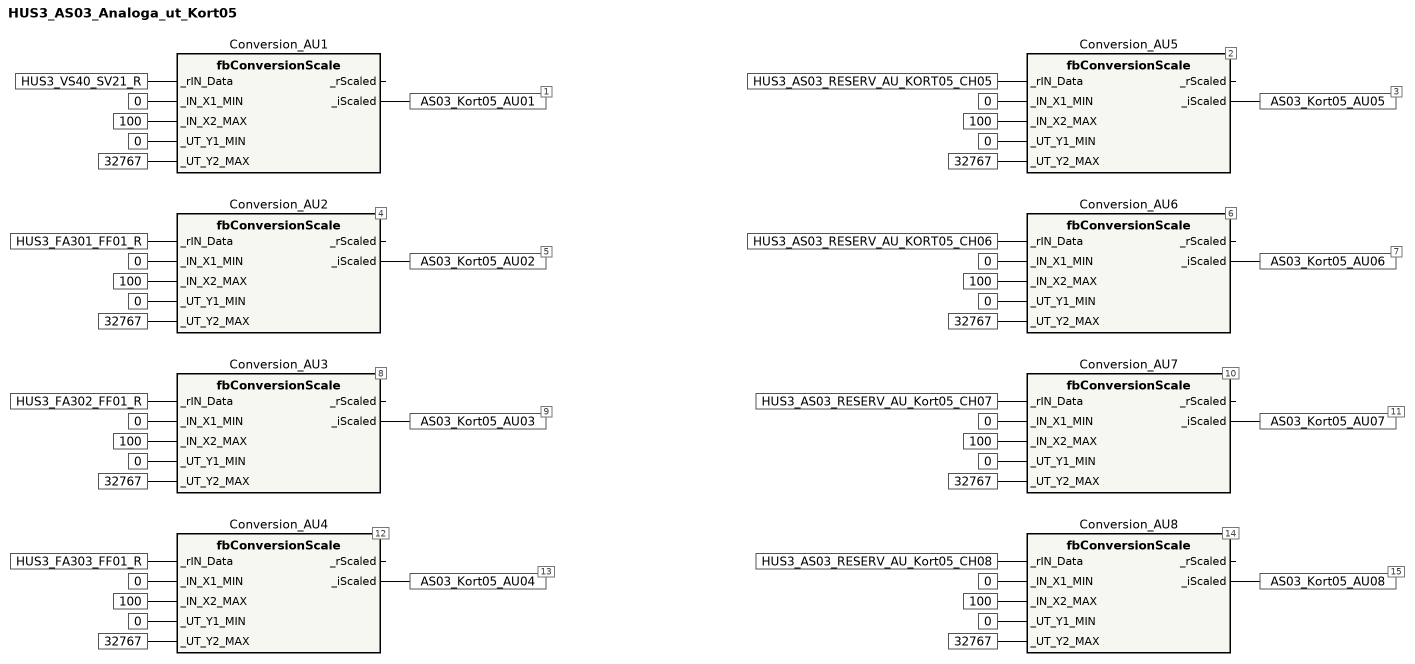
_CFC_ (* Continuous Function Chart, elements in execution order *)
#0 Conversion_AU1:fbConversionScale(_rIN_Data: HUS3_VS40_SV21_R, _IN_X1_MIN: 0, _IN_X2_MAX: 100, _UT_Y1_MIN: 0, _UT_Y2_MAX: 32767)
#1 AS03_Kort05_AU01 <= #0._iScaled
#2 Conversion_AU5:fbConversionScale(_rIN_Data: HUS3_AS03_RESERV_AU_KORT05_CH05, _IN_X1_MIN: 0, _IN_X2_MAX: 100, _UT_Y1_MIN: 0, _UT_Y2_MAX: 32767)
#3 AS03_Kort05_AU05 <= #2._iScaled
#4 Conversion_AU2:fbConversionScale(_rIN_Data: HUS3_FA301_FF01_R, _IN_X1_MIN: 0, _IN_X2_MAX: 100, _UT_Y1_MIN: 0, _UT_Y2_MAX: 32767)
#5 AS03_Kort05_AU02 <= #4._iScaled
#6 Conversion_AU6:fbConversionScale(_rIN_Data: HUS3_AS03_RESERV_AU_KORT05_CH06, _IN_X1_MIN: 0, _IN_X2_MAX: 100, _UT_Y1_MIN: 0, _UT_Y2_MAX: 32767)
#7 AS03_Kort05_AU06 <= #6._iScaled
#8 Conversion_AU3:fbConversionScale(_rIN_Data: HUS3_FA302_FF01_R, _IN_X1_MIN: 0, _IN_X2_MAX: 100, _UT_Y1_MIN: 0, _UT_Y2_MAX: 32767)
#9 AS03_Kort05_AU03 <= #8._iScaled
#10 Conversion_AU7:fbConversionScale(_rIN_Data: HUS3_AS03_RESERV_AU_Kort05_CH07, _IN_X1_MIN: 0, _IN_X2_MAX: 100, _UT_Y1_MIN: 0, _UT_Y2_MAX: 32767)
#11 AS03_Kort05_AU07 <= #10._iScaled
#12 Conversion_AU4:fbConversionScale(_rIN_Data: HUS3_FA303_FF01_R, _IN_X1_MIN: 0, _IN_X2_MAX: 100, _UT_Y1_MIN: 0, _UT_Y2_MAX: 32767)
#13 AS03_Kort05_AU04 <= #12._iScaled
#14 Conversion_AU8:fbConversionScale(_rIN_Data: HUS3_AS03_RESERV_AU_Kort05_CH08, _IN_X1_MIN: 0, _IN_X2_MAX: 100, _UT_Y1_MIN: 0, _UT_Y2_MAX: 32767)
#15 AS03_Kort05_AU08 <= #14._iScaled
_END_CFC_
(* the same logic as Structured Text *)
Conversion_AU1(_rIN_Data := HUS3_VS40_SV21_R, _IN_X1_MIN := 0, _IN_X2_MAX := 100, _UT_Y1_MIN := 0, _UT_Y2_MAX := 32767);
AS03_Kort05_AU01 := Conversion_AU1._iScaled;
Conversion_AU5(_rIN_Data := HUS3_AS03_RESERV_AU_KORT05_CH05, _IN_X1_MIN := 0, _IN_X2_MAX := 100, _UT_Y1_MIN := 0, _UT_Y2_MAX := 32767);
AS03_Kort05_AU05 := Conversion_AU5._iScaled;
Conversion_AU2(_rIN_Data := HUS3_FA301_FF01_R, _IN_X1_MIN := 0, _IN_X2_MAX := 100, _UT_Y1_MIN := 0, _UT_Y2_MAX := 32767);
AS03_Kort05_AU02 := Conversion_AU2._iScaled;
Conversion_AU6(_rIN_Data := HUS3_AS03_RESERV_AU_KORT05_CH06, _IN_X1_MIN := 0, _IN_X2_MAX := 100, _UT_Y1_MIN := 0, _UT_Y2_MAX := 32767);
AS03_Kort05_AU06 := Conversion_AU6._iScaled;
Conversion_AU3(_rIN_Data := HUS3_FA302_FF01_R, _IN_X1_MIN := 0, _IN_X2_MAX := 100, _UT_Y1_MIN := 0, _UT_Y2_MAX := 32767);
AS03_Kort05_AU03 := Conversion_AU3._iScaled;
Conversion_AU7(_rIN_Data := HUS3_AS03_RESERV_AU_Kort05_CH07, _IN_X1_MIN := 0, _IN_X2_MAX := 100, _UT_Y1_MIN := 0, _UT_Y2_MAX := 32767);
AS03_Kort05_AU07 := Conversion_AU7._iScaled;
Conversion_AU4(_rIN_Data := HUS3_FA303_FF01_R, _IN_X1_MIN := 0, _IN_X2_MAX := 100, _UT_Y1_MIN := 0, _UT_Y2_MAX := 32767);
AS03_Kort05_AU04 := Conversion_AU4._iScaled;
Conversion_AU8(_rIN_Data := HUS3_AS03_RESERV_AU_Kort05_CH08, _IN_X1_MIN := 0, _IN_X2_MAX := 100, _UT_Y1_MIN := 0, _UT_Y2_MAX := 32767);
AS03_Kort05_AU08 := Conversion_AU8._iScaled;
END_PROGRAM

(* POU _IOs_Uppdelat_per_skåp/HUS3_AL02/_IO/HUS3_AL02_IO_MAIN, CFC *)
PROGRAM HUS3_AL02_IO_MAIN
VAR
END_VAR
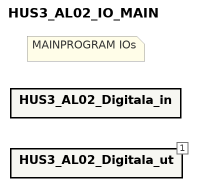
_CFC_ (* Continuous Function Chart, elements in execution order *)
(* MAINPROGRAM IOs *)
#0 HUS3_AL02_Digitala_in()
#1 HUS3_AL02_Digitala_ut()
_END_CFC_
(* the same logic as Structured Text *)
(* MAINPROGRAM IOs *)
HUS3_AL02_Digitala_in();
HUS3_AL02_Digitala_ut();
END_PROGRAM

(* POU _IOs_Uppdelat_per_skåp/HUS3_AL02/_IO/HUS3_AL02_Digitala_in, CFC *)
PROGRAM HUS3_AL02_Digitala_in

VAR


END_VAR
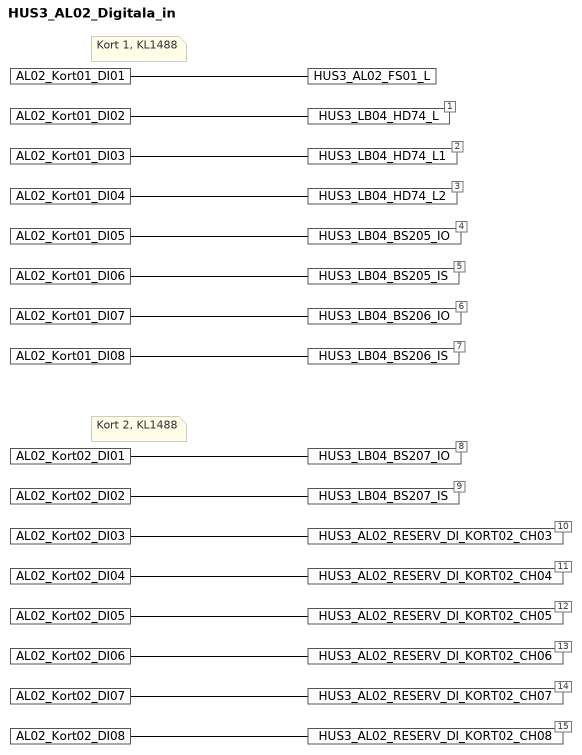
_CFC_ (* Continuous Function Chart, elements in execution order *)
(* Kort 2, KL1488 *)
(* Kort 1, KL1488 *)
#0 HUS3_AL02_FS01_L <= AL02_Kort01_DI01
#1 HUS3_LB04_HD74_L <= AL02_Kort01_DI02
#2 HUS3_LB04_HD74_L1 <= AL02_Kort01_DI03
#3 HUS3_LB04_HD74_L2 <= AL02_Kort01_DI04
#4 HUS3_LB04_BS205_IO <= AL02_Kort01_DI05
#5 HUS3_LB04_BS205_IS <= AL02_Kort01_DI06
#6 HUS3_LB04_BS206_IO <= AL02_Kort01_DI07
#7 HUS3_LB04_BS206_IS <= AL02_Kort01_DI08
#8 HUS3_LB04_BS207_IO <= AL02_Kort02_DI01
#9 HUS3_LB04_BS207_IS <= AL02_Kort02_DI02
#10 HUS3_AL02_RESERV_DI_KORT02_CH03 <= AL02_Kort02_DI03
#11 HUS3_AL02_RESERV_DI_KORT02_CH04 <= AL02_Kort02_DI04
#12 HUS3_AL02_RESERV_DI_KORT02_CH05 <= AL02_Kort02_DI05
#13 HUS3_AL02_RESERV_DI_KORT02_CH06 <= AL02_Kort02_DI06
#14 HUS3_AL02_RESERV_DI_KORT02_CH07 <= AL02_Kort02_DI07
#15 HUS3_AL02_RESERV_DI_KORT02_CH08 <= AL02_Kort02_DI08
_END_CFC_
(* the same logic as Structured Text *)
(* Kort 2, KL1488 *)
(* Kort 1, KL1488 *)
HUS3_AL02_FS01_L := AL02_Kort01_DI01;
HUS3_LB04_HD74_L := AL02_Kort01_DI02;
HUS3_LB04_HD74_L1 := AL02_Kort01_DI03;
HUS3_LB04_HD74_L2 := AL02_Kort01_DI04;
HUS3_LB04_BS205_IO := AL02_Kort01_DI05;
HUS3_LB04_BS205_IS := AL02_Kort01_DI06;
HUS3_LB04_BS206_IO := AL02_Kort01_DI07;
HUS3_LB04_BS206_IS := AL02_Kort01_DI08;
HUS3_LB04_BS207_IO := AL02_Kort02_DI01;
HUS3_LB04_BS207_IS := AL02_Kort02_DI02;
HUS3_AL02_RESERV_DI_KORT02_CH03 := AL02_Kort02_DI03;
HUS3_AL02_RESERV_DI_KORT02_CH04 := AL02_Kort02_DI04;
HUS3_AL02_RESERV_DI_KORT02_CH05 := AL02_Kort02_DI05;
HUS3_AL02_RESERV_DI_KORT02_CH06 := AL02_Kort02_DI06;
HUS3_AL02_RESERV_DI_KORT02_CH07 := AL02_Kort02_DI07;
HUS3_AL02_RESERV_DI_KORT02_CH08 := AL02_Kort02_DI08;
END_PROGRAM

(* POU _IOs_Uppdelat_per_skåp/HUS3_AL02/_IO/HUS3_AL02_Digitala_ut, CFC *)
PROGRAM HUS3_AL02_Digitala_ut


VAR
END_VAR
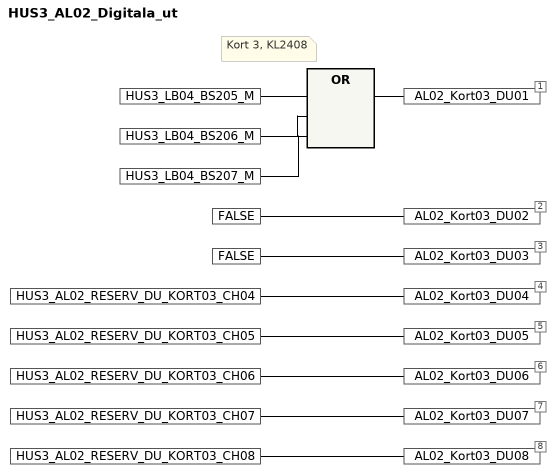
_CFC_ (* Continuous Function Chart, elements in execution order *)
(* Kort 3, KL2408 *)
#0 OR(HUS3_LB04_BS205_M, HUS3_LB04_BS206_M, HUS3_LB04_BS207_M)
#1 AL02_Kort03_DU01 <= #0
#2 AL02_Kort03_DU02 <= FALSE
#3 AL02_Kort03_DU03 <= FALSE
#4 AL02_Kort03_DU04 <= HUS3_AL02_RESERV_DU_KORT03_CH04
#5 AL02_Kort03_DU05 <= HUS3_AL02_RESERV_DU_KORT03_CH05
#6 AL02_Kort03_DU06 <= HUS3_AL02_RESERV_DU_KORT03_CH06
#7 AL02_Kort03_DU07 <= HUS3_AL02_RESERV_DU_KORT03_CH07
#8 AL02_Kort03_DU08 <= HUS3_AL02_RESERV_DU_KORT03_CH08
_END_CFC_
(* the same logic as Structured Text *)
(* Kort 3, KL2408 *)
AL02_Kort03_DU01 := HUS3_LB04_BS205_M OR HUS3_LB04_BS206_M OR HUS3_LB04_BS207_M;
AL02_Kort03_DU02 := FALSE;
AL02_Kort03_DU03 := FALSE;
AL02_Kort03_DU04 := HUS3_AL02_RESERV_DU_KORT03_CH04;
AL02_Kort03_DU05 := HUS3_AL02_RESERV_DU_KORT03_CH05;
AL02_Kort03_DU06 := HUS3_AL02_RESERV_DU_KORT03_CH06;
AL02_Kort03_DU07 := HUS3_AL02_RESERV_DU_KORT03_CH07;
AL02_Kort03_DU08 := HUS3_AL02_RESERV_DU_KORT03_CH08;
END_PROGRAM

(* POU _IOs_Uppdelat_per_skåp/HUS3_AL03/_IO/HUS3_AL03_IO_MAIN, CFC *)
PROGRAM HUS3_AL03_IO_MAIN
VAR
END_VAR
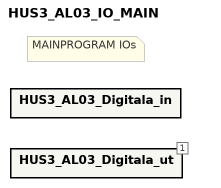
_CFC_ (* Continuous Function Chart, elements in execution order *)
(* MAINPROGRAM IOs *)
#0 HUS3_AL03_Digitala_in()
#1 HUS3_AL03_Digitala_ut()
_END_CFC_
(* the same logic as Structured Text *)
(* MAINPROGRAM IOs *)
HUS3_AL03_Digitala_in();
HUS3_AL03_Digitala_ut();
END_PROGRAM

(* POU _IOs_Uppdelat_per_skåp/HUS3_AL03/_IO/HUS3_AL03_Digitala_in, CFC *)
PROGRAM HUS3_AL03_Digitala_in

VAR


END_VAR
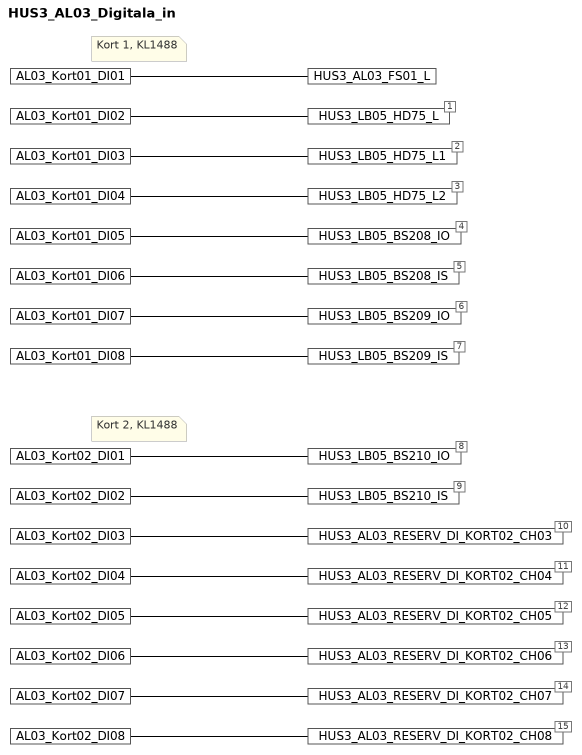
_CFC_ (* Continuous Function Chart, elements in execution order *)
(* Kort 1, KL1488 *)
(* Kort 2, KL1488 *)
#0 HUS3_AL03_FS01_L <= AL03_Kort01_DI01
#1 HUS3_LB05_HD75_L <= AL03_Kort01_DI02
#2 HUS3_LB05_HD75_L1 <= AL03_Kort01_DI03
#3 HUS3_LB05_HD75_L2 <= AL03_Kort01_DI04
#4 HUS3_LB05_BS208_IO <= AL03_Kort01_DI05
#5 HUS3_LB05_BS208_IS <= AL03_Kort01_DI06
#6 HUS3_LB05_BS209_IO <= AL03_Kort01_DI07
#7 HUS3_LB05_BS209_IS <= AL03_Kort01_DI08
#8 HUS3_LB05_BS210_IO <= AL03_Kort02_DI01
#9 HUS3_LB05_BS210_IS <= AL03_Kort02_DI02
#10 HUS3_AL03_RESERV_DI_KORT02_CH03 <= AL03_Kort02_DI03
#11 HUS3_AL03_RESERV_DI_KORT02_CH04 <= AL03_Kort02_DI04
#12 HUS3_AL03_RESERV_DI_KORT02_CH05 <= AL03_Kort02_DI05
#13 HUS3_AL03_RESERV_DI_KORT02_CH06 <= AL03_Kort02_DI06
#14 HUS3_AL03_RESERV_DI_KORT02_CH07 <= AL03_Kort02_DI07
#15 HUS3_AL03_RESERV_DI_KORT02_CH08 <= AL03_Kort02_DI08
_END_CFC_
(* the same logic as Structured Text *)
(* Kort 1, KL1488 *)
(* Kort 2, KL1488 *)
HUS3_AL03_FS01_L := AL03_Kort01_DI01;
HUS3_LB05_HD75_L := AL03_Kort01_DI02;
HUS3_LB05_HD75_L1 := AL03_Kort01_DI03;
HUS3_LB05_HD75_L2 := AL03_Kort01_DI04;
HUS3_LB05_BS208_IO := AL03_Kort01_DI05;
HUS3_LB05_BS208_IS := AL03_Kort01_DI06;
HUS3_LB05_BS209_IO := AL03_Kort01_DI07;
HUS3_LB05_BS209_IS := AL03_Kort01_DI08;
HUS3_LB05_BS210_IO := AL03_Kort02_DI01;
HUS3_LB05_BS210_IS := AL03_Kort02_DI02;
HUS3_AL03_RESERV_DI_KORT02_CH03 := AL03_Kort02_DI03;
HUS3_AL03_RESERV_DI_KORT02_CH04 := AL03_Kort02_DI04;
HUS3_AL03_RESERV_DI_KORT02_CH05 := AL03_Kort02_DI05;
HUS3_AL03_RESERV_DI_KORT02_CH06 := AL03_Kort02_DI06;
HUS3_AL03_RESERV_DI_KORT02_CH07 := AL03_Kort02_DI07;
HUS3_AL03_RESERV_DI_KORT02_CH08 := AL03_Kort02_DI08;
END_PROGRAM

(* POU _IOs_Uppdelat_per_skåp/HUS3_AL03/_IO/HUS3_AL03_Digitala_ut, CFC *)
PROGRAM HUS3_AL03_Digitala_ut


VAR
END_VAR
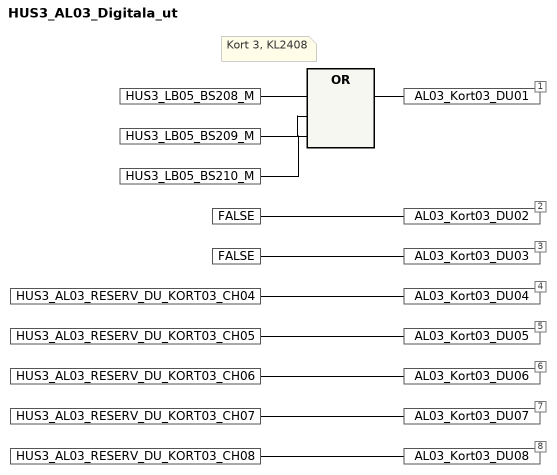
_CFC_ (* Continuous Function Chart, elements in execution order *)
(* Kort 3, KL2408 *)
#0 OR(HUS3_LB05_BS208_M, HUS3_LB05_BS209_M, HUS3_LB05_BS210_M)
#1 AL03_Kort03_DU01 <= #0
#2 AL03_Kort03_DU02 <= FALSE
#3 AL03_Kort03_DU03 <= FALSE
#4 AL03_Kort03_DU04 <= HUS3_AL03_RESERV_DU_KORT03_CH04
#5 AL03_Kort03_DU05 <= HUS3_AL03_RESERV_DU_KORT03_CH05
#6 AL03_Kort03_DU06 <= HUS3_AL03_RESERV_DU_KORT03_CH06
#7 AL03_Kort03_DU07 <= HUS3_AL03_RESERV_DU_KORT03_CH07
#8 AL03_Kort03_DU08 <= HUS3_AL03_RESERV_DU_KORT03_CH08
_END_CFC_
(* the same logic as Structured Text *)
(* Kort 3, KL2408 *)
AL03_Kort03_DU01 := HUS3_LB05_BS208_M OR HUS3_LB05_BS209_M OR HUS3_LB05_BS210_M;
AL03_Kort03_DU02 := FALSE;
AL03_Kort03_DU03 := FALSE;
AL03_Kort03_DU04 := HUS3_AL03_RESERV_DU_KORT03_CH04;
AL03_Kort03_DU05 := HUS3_AL03_RESERV_DU_KORT03_CH05;
AL03_Kort03_DU06 := HUS3_AL03_RESERV_DU_KORT03_CH06;
AL03_Kort03_DU07 := HUS3_AL03_RESERV_DU_KORT03_CH07;
AL03_Kort03_DU08 := HUS3_AL03_RESERV_DU_KORT03_CH08;
END_PROGRAM

(* POU SYSTEM/_Modbus TCP/HUS2_AS01_MODBUSTCP_MAIN, CFC *)
PROGRAM HUS2_AS01_MODBUSTCP_MAIN
VAR


END_VAR
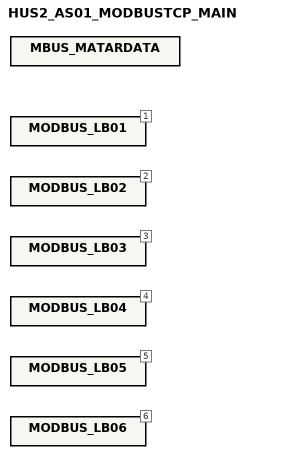
_CFC_ (* Continuous Function Chart, elements in execution order *)
#0 MBUS_MATARDATA()
#1 MODBUS_LB01()
#2 MODBUS_LB02()
#3 MODBUS_LB03()
#4 MODBUS_LB04()
#5 MODBUS_LB05()
#6 MODBUS_LB06()
_END_CFC_
(* the same logic as Structured Text *)
MBUS_MATARDATA();
MODBUS_LB01();
MODBUS_LB02();
MODBUS_LB03();
MODBUS_LB04();
MODBUS_LB05();
MODBUS_LB06();
END_PROGRAM

(* POU SYSTEM/_Modbus TCP/MBUS_MATARE/MBUS_MATARDATA, CFC *)
PROGRAM MBUS_MATARDATA
VAR

(* VP1-MQ41 *)
	Matare_VP1_MQ41: fbElvaco_GW_Integreringsverk;
	LC_Delay1: TON;
	bBusy1: BOOL;
	uiSlaveId					:BYTE:=16#FF;						(* Modbus slavadress *)

(* VV1-MQ41 *)
	Matare_VV1_MQ41: fbElvaco_GW_Integreringsverk;
	LC_Delay2: TON;
	bBusy2: BOOL;

(* VVC1-MQ41 *)
	Matare_VVC1_MQ41: fbElvaco_GW_Integreringsverk;
	LC_Delay3: TON;
	bBusy3: BOOL;

(* KV1-MF41 *)
	Matare_KV1_MF41: fbElvaco_GW_Flodesmatare;
	LC_Delay4: TON;
	bBusy4: BOOL;

(* KV1-MF42 *)
	Matare_KV1_MF42: fbElvaco_GW_Flodesmatare;
	LC_Delay5: TON;
	bBusy5: BOOL;



END_VAR
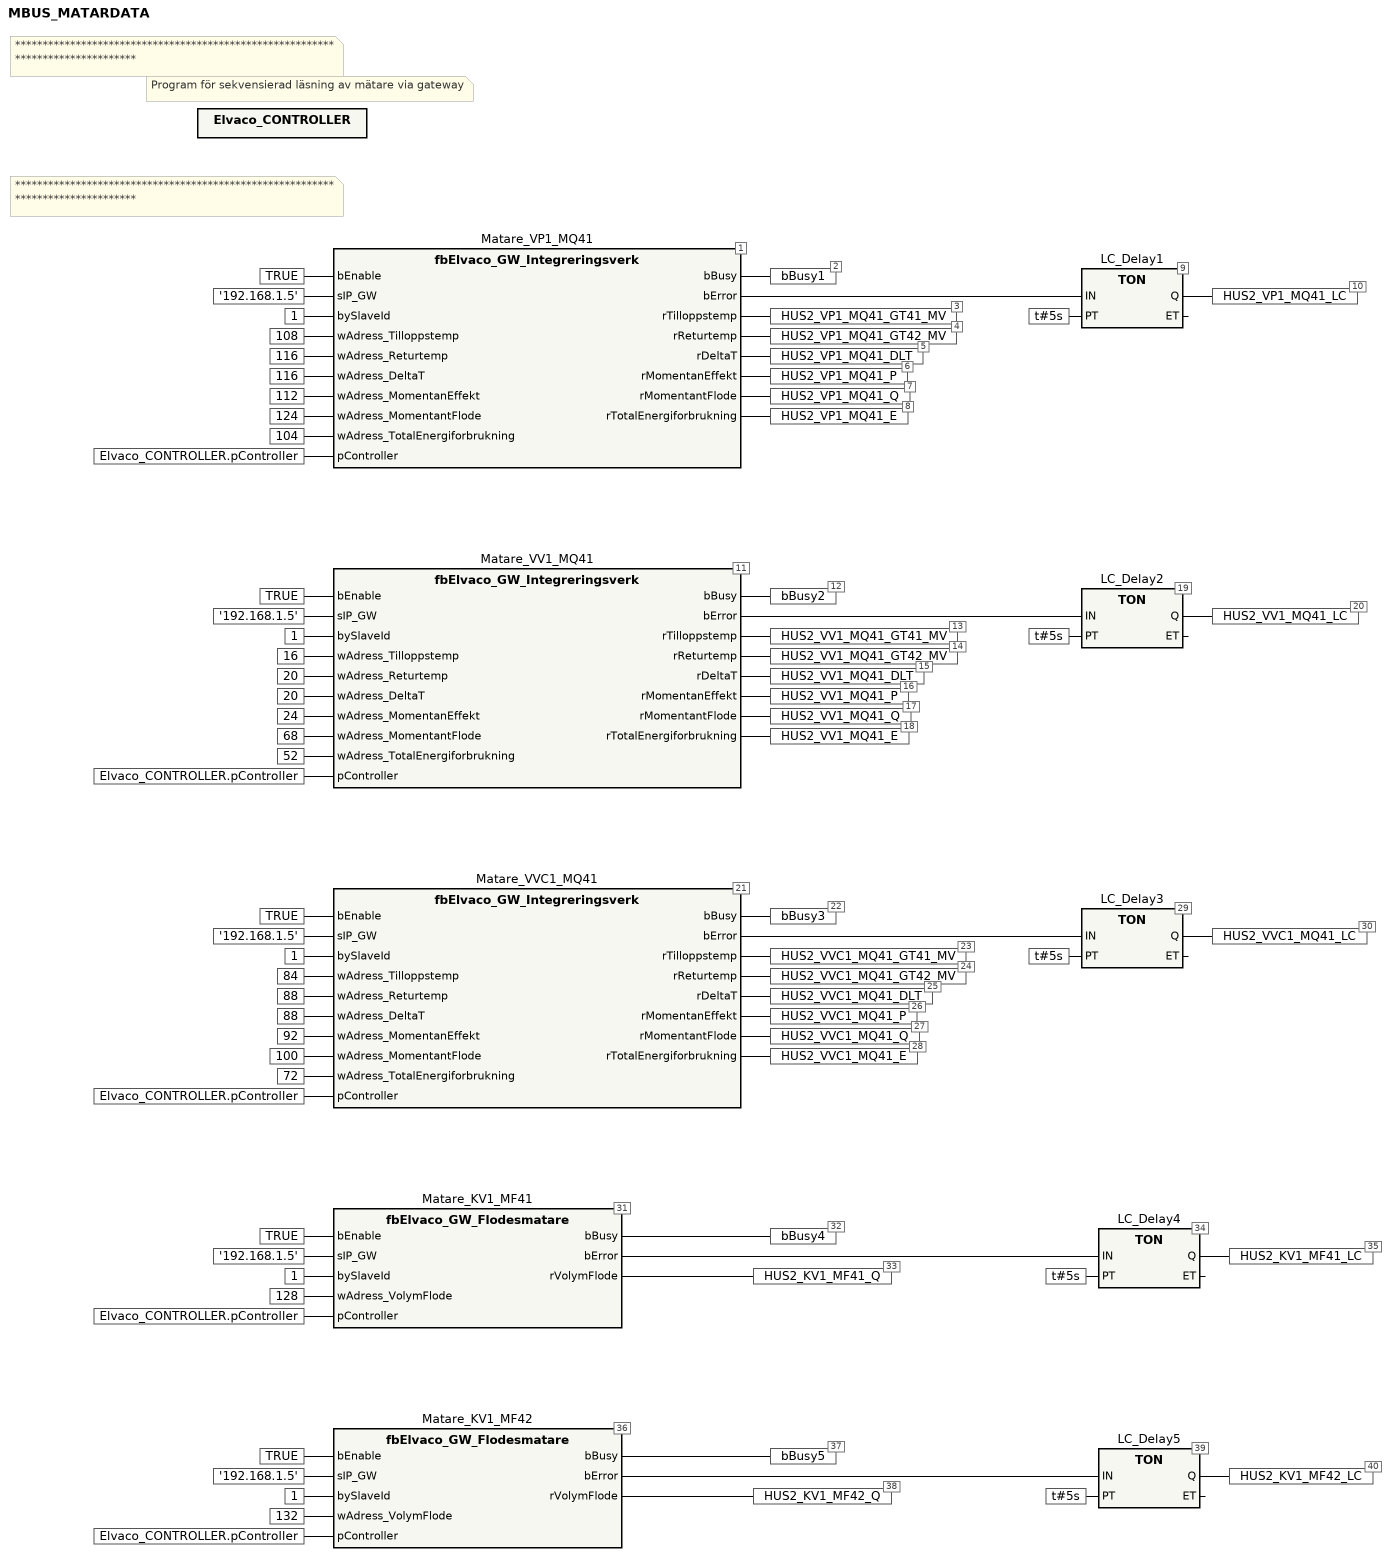
_CFC_ (* Continuous Function Chart, elements in execution order *)
(* ******************************************************************************** *)
(* ******************************************************************************** *)
(* Program för sekvensierad läsning av mätare via gateway *)
#0 Elvaco_CONTROLLER()
#1 Matare_VP1_MQ41:fbElvaco_GW_Integreringsverk(bEnable: TRUE, sIP_GW: '192.168.1.5', bySlaveId: 1, wAdress_Tilloppstemp: 108, wAdress_Returtemp: 116, wAdress_DeltaT: 116, wAdress_MomentanEffekt: 112, wAdress_MomentantFlode: 124, wAdress_TotalEnergiforbrukning: 104, pController: Elvaco_CONTROLLER.pController)
#2 bBusy1 <= #1.bBusy
#3 HUS2_VP1_MQ41_GT41_MV <= #1.rTilloppstemp
#4 HUS2_VP1_MQ41_GT42_MV <= #1.rReturtemp
#5 HUS2_VP1_MQ41_DLT <= #1.rDeltaT
#6 HUS2_VP1_MQ41_P <= #1.rMomentanEffekt
#7 HUS2_VP1_MQ41_Q <= #1.rMomentantFlode
#8 HUS2_VP1_MQ41_E <= #1.rTotalEnergiforbrukning
#9 LC_Delay1:TON(IN: #1.bError, PT: t#5s)
#10 HUS2_VP1_MQ41_LC <= #9.Q
#11 Matare_VV1_MQ41:fbElvaco_GW_Integreringsverk(bEnable: TRUE, sIP_GW: '192.168.1.5', bySlaveId: 1, wAdress_Tilloppstemp: 16, wAdress_Returtemp: 20, wAdress_DeltaT: 20, wAdress_MomentanEffekt: 24, wAdress_MomentantFlode: 68, wAdress_TotalEnergiforbrukning: 52, pController: Elvaco_CONTROLLER.pController)
#12 bBusy2 <= #11.bBusy
#13 HUS2_VV1_MQ41_GT41_MV <= #11.rTilloppstemp
#14 HUS2_VV1_MQ41_GT42_MV <= #11.rReturtemp
#15 HUS2_VV1_MQ41_DLT <= #11.rDeltaT
#16 HUS2_VV1_MQ41_P <= #11.rMomentanEffekt
#17 HUS2_VV1_MQ41_Q <= #11.rMomentantFlode
#18 HUS2_VV1_MQ41_E <= #11.rTotalEnergiforbrukning
#19 LC_Delay2:TON(IN: #11.bError, PT: t#5s)
#20 HUS2_VV1_MQ41_LC <= #19.Q
#21 Matare_VVC1_MQ41:fbElvaco_GW_Integreringsverk(bEnable: TRUE, sIP_GW: '192.168.1.5', bySlaveId: 1, wAdress_Tilloppstemp: 84, wAdress_Returtemp: 88, wAdress_DeltaT: 88, wAdress_MomentanEffekt: 92, wAdress_MomentantFlode: 100, wAdress_TotalEnergiforbrukning: 72, pController: Elvaco_CONTROLLER.pController)
#22 bBusy3 <= #21.bBusy
#23 HUS2_VVC1_MQ41_GT41_MV <= #21.rTilloppstemp
#24 HUS2_VVC1_MQ41_GT42_MV <= #21.rReturtemp
#25 HUS2_VVC1_MQ41_DLT <= #21.rDeltaT
#26 HUS2_VVC1_MQ41_P <= #21.rMomentanEffekt
#27 HUS2_VVC1_MQ41_Q <= #21.rMomentantFlode
#28 HUS2_VVC1_MQ41_E <= #21.rTotalEnergiforbrukning
#29 LC_Delay3:TON(IN: #21.bError, PT: t#5s)
#30 HUS2_VVC1_MQ41_LC <= #29.Q
#31 Matare_KV1_MF41:fbElvaco_GW_Flodesmatare(bEnable: TRUE, sIP_GW: '192.168.1.5', bySlaveId: 1, wAdress_VolymFlode: 128, pController: Elvaco_CONTROLLER.pController)
#32 bBusy4 <= #31.bBusy
#33 HUS2_KV1_MF41_Q <= #31.rVolymFlode
#34 LC_Delay4:TON(IN: #31.bError, PT: t#5s)
#35 HUS2_KV1_MF41_LC <= #34.Q
#36 Matare_KV1_MF42:fbElvaco_GW_Flodesmatare(bEnable: TRUE, sIP_GW: '192.168.1.5', bySlaveId: 1, wAdress_VolymFlode: 132, pController: Elvaco_CONTROLLER.pController)
#37 bBusy5 <= #36.bBusy
#38 HUS2_KV1_MF42_Q <= #36.rVolymFlode
#39 LC_Delay5:TON(IN: #36.bError, PT: t#5s)
#40 HUS2_KV1_MF42_LC <= #39.Q
_END_CFC_
(* the same logic as Structured Text *)
(* ******************************************************************************** *)
(* ******************************************************************************** *)
(* Program för sekvensierad läsning av mätare via gateway *)
Elvaco_CONTROLLER();
Matare_VP1_MQ41(bEnable := TRUE, sIP_GW := '192.168.1.5', bySlaveId := 1, wAdress_Tilloppstemp := 108, wAdress_Returtemp := 116, wAdress_DeltaT := 116, wAdress_MomentanEffekt := 112, wAdress_MomentantFlode := 124, wAdress_TotalEnergiforbrukning := 104, pController := Elvaco_CONTROLLER.pController);
bBusy1 := Matare_VP1_MQ41.bBusy;
HUS2_VP1_MQ41_GT41_MV := Matare_VP1_MQ41.rTilloppstemp;
HUS2_VP1_MQ41_GT42_MV := Matare_VP1_MQ41.rReturtemp;
HUS2_VP1_MQ41_DLT := Matare_VP1_MQ41.rDeltaT;
HUS2_VP1_MQ41_P := Matare_VP1_MQ41.rMomentanEffekt;
HUS2_VP1_MQ41_Q := Matare_VP1_MQ41.rMomentantFlode;
HUS2_VP1_MQ41_E := Matare_VP1_MQ41.rTotalEnergiforbrukning;
LC_Delay1(IN := Matare_VP1_MQ41.bError, PT := t#5s);
HUS2_VP1_MQ41_LC := LC_Delay1.Q;
Matare_VV1_MQ41(bEnable := TRUE, sIP_GW := '192.168.1.5', bySlaveId := 1, wAdress_Tilloppstemp := 16, wAdress_Returtemp := 20, wAdress_DeltaT := 20, wAdress_MomentanEffekt := 24, wAdress_MomentantFlode := 68, wAdress_TotalEnergiforbrukning := 52, pController := Elvaco_CONTROLLER.pController);
bBusy2 := Matare_VV1_MQ41.bBusy;
HUS2_VV1_MQ41_GT41_MV := Matare_VV1_MQ41.rTilloppstemp;
HUS2_VV1_MQ41_GT42_MV := Matare_VV1_MQ41.rReturtemp;
HUS2_VV1_MQ41_DLT := Matare_VV1_MQ41.rDeltaT;
HUS2_VV1_MQ41_P := Matare_VV1_MQ41.rMomentanEffekt;
HUS2_VV1_MQ41_Q := Matare_VV1_MQ41.rMomentantFlode;
HUS2_VV1_MQ41_E := Matare_VV1_MQ41.rTotalEnergiforbrukning;
LC_Delay2(IN := Matare_VV1_MQ41.bError, PT := t#5s);
HUS2_VV1_MQ41_LC := LC_Delay2.Q;
Matare_VVC1_MQ41(bEnable := TRUE, sIP_GW := '192.168.1.5', bySlaveId := 1, wAdress_Tilloppstemp := 84, wAdress_Returtemp := 88, wAdress_DeltaT := 88, wAdress_MomentanEffekt := 92, wAdress_MomentantFlode := 100, wAdress_TotalEnergiforbrukning := 72, pController := Elvaco_CONTROLLER.pController);
bBusy3 := Matare_VVC1_MQ41.bBusy;
HUS2_VVC1_MQ41_GT41_MV := Matare_VVC1_MQ41.rTilloppstemp;
HUS2_VVC1_MQ41_GT42_MV := Matare_VVC1_MQ41.rReturtemp;
HUS2_VVC1_MQ41_DLT := Matare_VVC1_MQ41.rDeltaT;
HUS2_VVC1_MQ41_P := Matare_VVC1_MQ41.rMomentanEffekt;
HUS2_VVC1_MQ41_Q := Matare_VVC1_MQ41.rMomentantFlode;
HUS2_VVC1_MQ41_E := Matare_VVC1_MQ41.rTotalEnergiforbrukning;
LC_Delay3(IN := Matare_VVC1_MQ41.bError, PT := t#5s);
HUS2_VVC1_MQ41_LC := LC_Delay3.Q;
Matare_KV1_MF41(bEnable := TRUE, sIP_GW := '192.168.1.5', bySlaveId := 1, wAdress_VolymFlode := 128, pController := Elvaco_CONTROLLER.pController);
bBusy4 := Matare_KV1_MF41.bBusy;
HUS2_KV1_MF41_Q := Matare_KV1_MF41.rVolymFlode;
LC_Delay4(IN := Matare_KV1_MF41.bError, PT := t#5s);
HUS2_KV1_MF41_LC := LC_Delay4.Q;
Matare_KV1_MF42(bEnable := TRUE, sIP_GW := '192.168.1.5', bySlaveId := 1, wAdress_VolymFlode := 132, pController := Elvaco_CONTROLLER.pController);
bBusy5 := Matare_KV1_MF42.bBusy;
HUS2_KV1_MF42_Q := Matare_KV1_MF42.rVolymFlode;
LC_Delay5(IN := Matare_KV1_MF42.bError, PT := t#5s);
HUS2_KV1_MF42_LC := LC_Delay5.Q;
END_PROGRAM

(* POU xEgna Funktionsblock/Modbus/Elvaco/fbElvaco_GW_Integreringsverk, ST *)
FUNCTION_BLOCK fbElvaco_GW_Integreringsverk

VAR
	MB_ReadRegs 				:FB_MBReadRegs;				(* Modbusmaster read holding registers *)
	iDx								:INT:= 0;							(* Index för sekvensen *)

(* Variables used for generic handling *)
	bReturnAfterAction	 		:BOOL;
	bInit 							:BOOL := TRUE;
	nState 							:INT;
	iGenericID 						:INT;

(* Läst data*)

	rTilloppstemp_read				:REAL;							(* Grader Celsius *)
	rReturtemp_read					:REAL;							(* Grader Celsius *)
	rDeltaT_read						:REAL;							(* Grader Kelvin *)
	rMomentanEffekt_read			:REAL;							(* kW *)
	rMomentantFlode_read			:REAL;							(* m3/h *)
	rTotalEnergiforbrukning_read		:REAL;							(* MWh *)


END_VAR
VAR_INPUT
	bEnable								:BOOL;							(* Starta läsning *)
	sIP_GW								:STRING;							(* IP-adress Elvaco gateway *)
	bySlaveId								:BYTE;								(* M-busslavens ID *)

	wAdress_Tilloppstemp				:WORD;
	wAdress_Returtemp					:WORD;
	wAdress_DeltaT						:WORD;
	wAdress_MomentanEffekt			:WORD;
	wAdress_MomentantFlode			:WORD;
	wAdress_TotalEnergiforbrukning		:WORD;



(*Skicka in en pekare till controllerstrukten *)
	pController					:POINTER TO ST_Elvaco_CONTROLLER;	(* Pekare till strukturen *)

END_VAR
VAR_OUTPUT
	bBusy							:BOOL;
	bError							:BOOL;						(* Vi har ett fel *)

	rTilloppstemp					:REAL;							(* Grader Celsius *)
	rReturtemp						:REAL;							(* Grader Celsius *)
	rDeltaT						:REAL;							(* Grader Kelvin *)
	rMomentanEffekt				:REAL;							(* kW *)
	rMomentantFlode				:REAL;							(* m3/h *)
	rTotalEnergiforbrukning		:REAL;							(* MWh *)


END_VAR
actGenericHandling();
IF bReturnAfterAction THEN
	RETURN;
END_IF


CASE iDx OF

0:(*Vänta på start*)
		pController^.bUnitIsBusy:=TRUE;
		pController^.bUnitIsDone:=FALSE;
		bBusy:=TRUE;
		iDx := 10;



10:(*Läs Holding Registers *)
	MB_ReadRegs(sIPAddr		:= sIP_GW,
					nUnitID		:= bySlaveId ,
					nTCPPort		:=502,
					nQuantity		:= 2,
					nMBAddR		:= wAdress_Tilloppstemp,
					cbLength		:= SIZEOF(rTilloppstemp_read),
					pDestAddr	:= ADR(rTilloppstemp_read),
					bExecute		:= TRUE ,
					tTimeout		:= T#1s ,
					bBusy=> ,
					bError=> ,
					nErrId=> ,
					cbRead=> );

	IF NOT MB_ReadRegs.bBusy AND NOT MB_ReadRegs.bError THEN
		MB_ReadRegs(bExecute:=FALSE);
		bError := FALSE;
		iDx := 15;
	ELSIF MB_ReadRegs.bError THEN
		MB_ReadRegs(bExecute:=FALSE);
		iDx := 999;
	END_IF


15:(*Läs Holding Registers *)
	MB_ReadRegs(sIPAddr		:= sIP_GW,
					nUnitID		:= bySlaveId ,
					nTCPPort		:=502,
					nQuantity		:= 2,
					nMBAddR		:= wAdress_Returtemp,
					cbLength		:= SIZEOF(rReturtemp_read),
					pDestAddr	:= ADR(rReturtemp_read),
					bExecute		:= TRUE ,
					tTimeout		:= T#1s ,
					bBusy=> ,
					bError=> ,
					nErrId=> ,
					cbRead=> );

	IF NOT MB_ReadRegs.bBusy AND NOT MB_ReadRegs.bError THEN
		MB_ReadRegs(bExecute:=FALSE);
		bError := FALSE;
		iDx := 20;
	ELSIF MB_ReadRegs.bError THEN
		MB_ReadRegs(bExecute:=FALSE);
		iDx := 999;
	END_IF


20:(*Läs Holding Registers *)
	MB_ReadRegs(sIPAddr		:= sIP_GW,
					nUnitID		:= bySlaveId ,
					nTCPPort		:=502,
					nQuantity		:= 2,
					nMBAddR		:= wAdress_DeltaT,
					cbLength		:= SIZEOF(rDeltaT_read),
					pDestAddr	:= ADR(rDeltaT_read),
					bExecute		:= TRUE ,
					tTimeout		:= T#1s ,
					bBusy=> ,
					bError=> ,
					nErrId=> ,
					cbRead=> );

	IF NOT MB_ReadRegs.bBusy AND NOT MB_ReadRegs.bError THEN
		MB_ReadRegs(bExecute:=FALSE);
		bError := FALSE;
		iDx := 25;
	ELSIF MB_ReadRegs.bError THEN
		MB_ReadRegs(bExecute:=FALSE);
		iDx := 999;
	END_IF


25:(*Läs Holding Registers *)
	MB_ReadRegs(sIPAddr		:= sIP_GW,
					nUnitID		:= bySlaveId ,
					nTCPPort		:=502,
					nQuantity		:= 2,
					nMBAddR		:= wAdress_MomentanEffekt,
					cbLength		:= SIZEOF(rMomentanEffekt_read),
					pDestAddr	:= ADR(rMomentanEffekt_read),
					bExecute		:= TRUE ,
					tTimeout		:= T#1s ,
					bBusy=> ,
					bError=> ,
					nErrId=> ,
					cbRead=> );

	IF NOT MB_ReadRegs.bBusy AND NOT MB_ReadRegs.bError THEN
		MB_ReadRegs(bExecute:=FALSE);
		bError := FALSE;
		iDx := 30;
	ELSIF MB_ReadRegs.bError THEN
		MB_ReadRegs(bExecute:=FALSE);
		iDx := 999;
	END_IF


30:(*Läs Holding Registers *)
	MB_ReadRegs(sIPAddr		:= sIP_GW,
					nUnitID		:= bySlaveId ,
					nTCPPort		:=502,
					nQuantity		:= 2,
					nMBAddR		:= wAdress_MomentantFlode,
					cbLength		:= SIZEOF(rMomentantFlode_read),
					pDestAddr	:= ADR(rMomentantFlode_read),
					bExecute		:= TRUE ,
					tTimeout		:= T#1s ,
					bBusy=> ,
					bError=> ,
					nErrId=> ,
					cbRead=> );

	IF NOT MB_ReadRegs.bBusy AND NOT MB_ReadRegs.bError THEN
		MB_ReadRegs(bExecute:=FALSE);
		bError := FALSE;
		iDx := 35;
	ELSIF MB_ReadRegs.bError THEN
		MB_ReadRegs(bExecute:=FALSE);
		iDx := 999;
	END_IF


35:(*Läs Holding Registers *)
	MB_ReadRegs(sIPAddr		:= sIP_GW,
					nUnitID		:= bySlaveId ,
					nTCPPort		:=502,
					nQuantity		:= 2,
					nMBAddR		:= wAdress_TotalEnergiforbrukning,
					cbLength		:= SIZEOF(rTotalEnergiforbrukning_read),
					pDestAddr	:= ADR(rTotalEnergiforbrukning_read),
					bExecute		:= TRUE ,
					tTimeout		:= T#1s ,
					bBusy=> ,
					bError=> ,
					nErrId=> ,
					cbRead=> );

	IF NOT MB_ReadRegs.bBusy AND NOT MB_ReadRegs.bError THEN
		MB_ReadRegs(bExecute:=FALSE);
		bError := FALSE;
		iDx := 100;
	ELSIF MB_ReadRegs.bError THEN
		MB_ReadRegs(bExecute:=FALSE);
		iDx := 999;
	END_IF



	(*Anropa actions och kontrollera om skrivning behövs*)
100:	fbElvaco_GW_Integreringsverk.actCalculateData;


888: (*DONE*)
	pController^.bUnitIsBusy:=FALSE;
	pController^.bUnitIsDone:=TRUE;
	bBusy:=FALSE;
	iDx := 0;


999: (*ERROR*)
	pController^.bUnitIsBusy:=FALSE;
	pController^.bUnitIsDone:=TRUE;
	MB_ReadRegs(bExecute := FALSE);
	bError := TRUE;
	bBusy:=FALSE;
	iDx := 0;


END_CASE
END_FUNCTION_BLOCK
ACTION actCalculateData:
(*Beräkning/konvertering av signaler till utgång*)



(* MÄTVÄRDEN & UTSIGNALER *)

	rTilloppstemp:=						rTilloppstemp_read*0.01;
	rReturtemp:=							rReturtemp_read*0.01;
	rDeltaT:=								(rTilloppstemp-rReturtemp);
	rMomentanEffekt:=					rMomentanEffekt_read*0.00001;
	rMomentantFlode:=					rMomentantFlode_read*0.01;
	rTotalEnergiforbrukning:=				rTotalEnergiforbrukning_read*0.00000001;


(* GÅ TILL NÄSTA STEG *)
	iDx := 888;
END_ACTION
ACTION actGenericHandling:
(* DO NOT ALTER/REMOVE *)
bReturnAfterAction:=TRUE;
(* Exit if invalid controller pointer *)
IF pController=0 THEN
	RETURN;
END_IF

(* One time initialisation *)
IF bInit THEN
	(* "Register" this block in the controller using the incremental index *)
	pController^.iNoUnits:=pController^.iNoUnits+1;
	(* Assign the generic ID of this unit *)
	iGenericID:=pController^.iNoUnits;
	(* Init done *)
	bInit:=FALSE;
END_IF

(* Exit if controller working ID doesn't match the unit ID *)
IF pController^.iWorkingUnitId<>iGenericID THEN
	RETURN;
END_IF

(* If unit isn't enabled then signal that we're done as soon as it's our turn *)
IF NOT bEnable THEN
	pController^.bUnitIsDone:=TRUE;
	pController^.bUnitIsBusy:=FALSE;
	RETURN;
END_IF

(* The code managed to get here without returning, that means we should execute the rest of the function block as well *)
bReturnAfterAction:=FALSE;
END_ACTION

(* POU xEgna Funktionsblock/Modbus/Elvaco/fbElvaco_GW_Flodesmatare, ST *)
FUNCTION_BLOCK fbElvaco_GW_Flodesmatare

VAR
	MB_ReadRegs 				:FB_MBReadRegs;				(* Modbusmaster read holding registers *)
	iDx								:INT:= 0;							(* Index för sekvensen *)

(* Variables used for generic handling *)
	bReturnAfterAction	 		:BOOL;
	bInit 							:BOOL := TRUE;
	nState 							:INT;
	iGenericID 						:INT;

(* Läst data*)

	wVolymFlode_read				:WORD;							(* m3 *)
	rVolymFlode_read					:REAL;								(* m3 *)

END_VAR
VAR_INPUT
	bEnable								:BOOL;							(* Starta läsning *)
	sIP_GW								:STRING;							(* IP-adress Elvaco gateway *)
	bySlaveId								:BYTE;								(* M-busslavens ID *)
	wAdress_VolymFlode					:WORD;


(*Skicka in en pekare till controllerstrukten *)
	pController					:POINTER TO ST_Elvaco_CONTROLLER;	(* Pekare till strukturen *)

END_VAR
VAR_OUTPUT
	bBusy							:BOOL;
	bError							:BOOL;						(* Vi har ett fel *)

	rVolymFlode					:REAL;							(* m3 *)


END_VAR
actGenericHandling();
IF bReturnAfterAction THEN
	RETURN;
END_IF


CASE iDx OF

0:(*Vänta på start*)
		pController^.bUnitIsBusy:=TRUE;
		pController^.bUnitIsDone:=FALSE;
		bBusy:=TRUE;
		iDx := 5;


5:(*Läs Holding Registers *)
	MB_ReadRegs(sIPAddr		:= sIP_GW,
					nTCPPort		:=502,
					nUnitID		:= bySlaveId,
					nQuantity		:= 2,
					nMBAddR		:= wAdress_VolymFlode,
					cbLength		:= SIZEOF(rVolymFlode_read),
					pDestAddr	:= ADR(rVolymFlode_read),
					bExecute		:= TRUE ,
					tTimeout		:= T#2s ,
					bBusy=> ,
					bError=> ,
					nErrId=> ,
					cbRead=> );

	IF NOT MB_ReadRegs.bBusy AND NOT MB_ReadRegs.bError THEN
		MB_ReadRegs(bExecute:=FALSE);
		bError := FALSE;

	rVolymFlode:=	rVolymFlode_read*0.01;

		iDx := 888;
	ELSIF MB_ReadRegs.bError THEN
		MB_ReadRegs(bExecute:=FALSE);
		iDx := 999;
	END_IF


888: (*DONE*)
	pController^.bUnitIsBusy:=FALSE;
	pController^.bUnitIsDone:=TRUE;
	bBusy:=FALSE;
	iDx := 0;


999: (*ERROR*)
	pController^.bUnitIsBusy:=FALSE;
	pController^.bUnitIsDone:=TRUE;
	MB_ReadRegs(bExecute := FALSE);
	bError := TRUE;
	bBusy:=FALSE;
	iDx := 0;


END_CASE
END_FUNCTION_BLOCK
ACTION actGenericHandling:
(* DO NOT ALTER/REMOVE *)
bReturnAfterAction:=TRUE;
(* Exit if invalid controller pointer *)
IF pController=0 THEN
	RETURN;
END_IF

(* One time initialisation *)
IF bInit THEN
	(* "Register" this block in the controller using the incremental index *)
	pController^.iNoUnits:=pController^.iNoUnits+1;
	(* Assign the generic ID of this unit *)
	iGenericID:=pController^.iNoUnits;
	(* Init done *)
	bInit:=FALSE;
END_IF

(* Exit if controller working ID doesn't match the unit ID *)
IF pController^.iWorkingUnitId<>iGenericID THEN
	RETURN;
END_IF

(* If unit isn't enabled then signal that we're done as soon as it's our turn *)
IF NOT bEnable THEN
	pController^.bUnitIsDone:=TRUE;
	pController^.bUnitIsBusy:=FALSE;
	RETURN;
END_IF

(* The code managed to get here without returning, that means we should execute the rest of the function block as well *)
bReturnAfterAction:=FALSE;
END_ACTION

(* POU SYSTEM/_Modbus TCP/MBUS_MATARE/Elvaco_CONTROLLER, ST *)
PROGRAM Elvaco_CONTROLLER
VAR_OUTPUT

END_VAR
VAR
	stController			: ST_Elvaco_CONTROLLER:=(iWorkingUnitId:=1);
	pController			: POINTER TO ST_Elvaco_CONTROLLER;
END_VAR
(* DO NOT CHANGE ANYTHING IN THIS CODE *)

(* Output the pointer to this controller*)
pController := ADR(stController);

(* Do any units exist? *)
IF stController.iNoUnits>0 THEN
	(* Is the current unit done? *)
	IF stController.bUnitIsDone  THEN
		(* Yes, reset the done flag and increase the unit ID counter *)
		stController.bUnitIsDone:=FALSE;
		stController.iWorkingUnitId:=stController.iWorkingUnitId+1;
		(*Handle rollover of the unit ID counter *)
		IF stController.iWorkingUnitId>stController.iNoUnits THEN
			stController.iWorkingUnitId:=1;
		END_IF
	END_IF
END_IF
END_PROGRAM

(* POU SYSTEM/_Modbus TCP/GOLD_AGGREGAT/MODBUS_LB01, CFC *)
PROGRAM MODBUS_LB01
VAR

	KOMFEL_DELAY: fbDelayedAlarmMinutes;

(*LB01*)
	LB01_MODBUS: fbSwegonGOLD_v1;
	bEnableRead			:BOOL:=TRUE;
	bEnableWrite			:BOOL:=TRUE;			(*SÄTT TILL INITIAL TRUE VID DRIFTSÄTTNING*)
	bError					:BOOL;
	bBusy					:BOOL;

	rDUMMY_GT11_MIN1	:REAL;
	rDUMMY_GT11_MAX1	:REAL;
	rDUMMY_GT41_BV1		:REAL;
	rDUMMY_GP11_LOW1	:REAL;
	rDUMMY_GP12_LOW1	:REAL;
	bLB01_TILL				:BOOL;

END_VAR
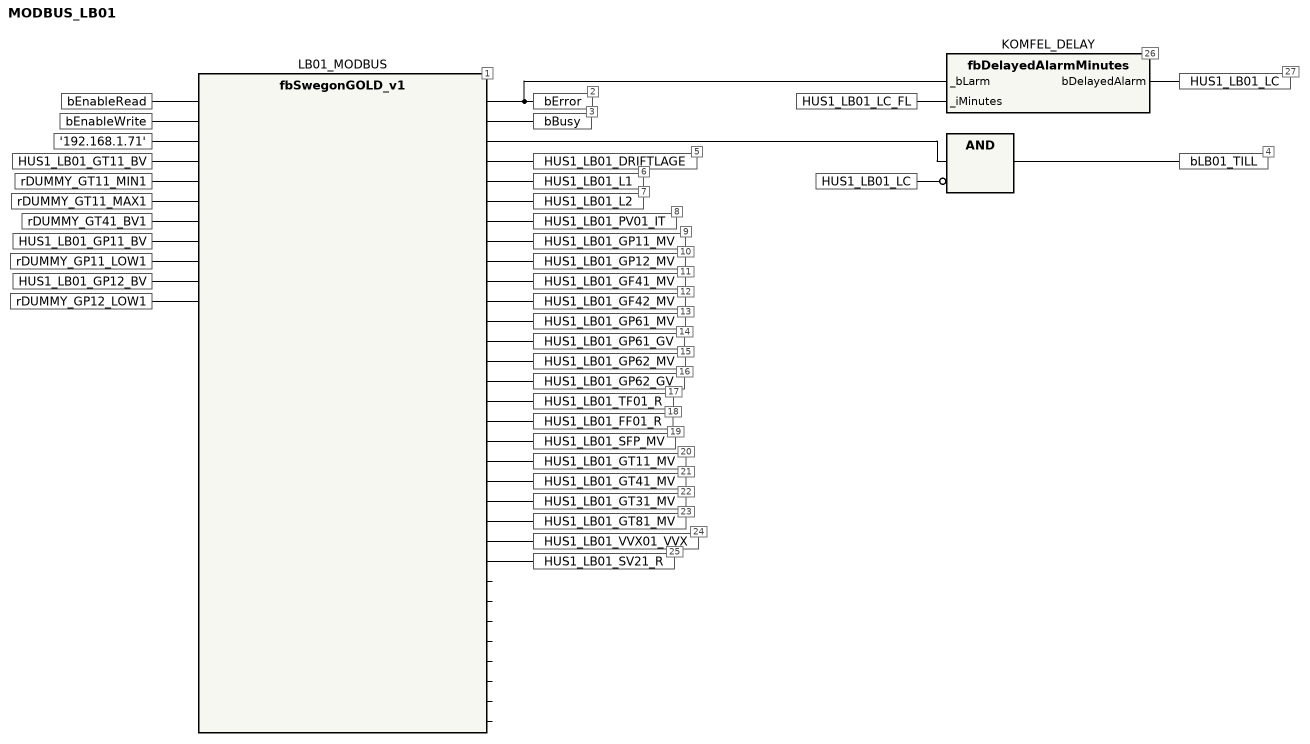
_CFC_ (* Continuous Function Chart, elements in execution order *)
#0 AND(#1.out 3, NOT HUS1_LB01_LC)
#1 LB01_MODBUS:fbSwegonGOLD_v1(bEnableRead, bEnableWrite, '192.168.1.71', HUS1_LB01_GT11_BV, rDUMMY_GT11_MIN1, rDUMMY_GT11_MAX1, rDUMMY_GT41_BV1, HUS1_LB01_GP11_BV, rDUMMY_GP11_LOW1, HUS1_LB01_GP12_BV, rDUMMY_GP12_LOW1)
#2 bError <= #1.out 1
#3 bBusy <= #1.out 2
#4 bLB01_TILL <= #0
#5 HUS1_LB01_DRIFTLAGE <= #1.out 4
#6 HUS1_LB01_L1 <= #1.out 5
#7 HUS1_LB01_L2 <= #1.out 6
#8 HUS1_LB01_PV01_IT <= #1.out 7
#9 HUS1_LB01_GP11_MV <= #1.out 8
#10 HUS1_LB01_GP12_MV <= #1.out 9
#11 HUS1_LB01_GF41_MV <= #1.out 10
#12 HUS1_LB01_GF42_MV <= #1.out 11
#13 HUS1_LB01_GP61_MV <= #1.out 12
#14 HUS1_LB01_GP61_GV <= #1.out 13
#15 HUS1_LB01_GP62_MV <= #1.out 14
#16 HUS1_LB01_GP62_GV <= #1.out 15
#17 HUS1_LB01_TF01_R <= #1.out 16
#18 HUS1_LB01_FF01_R <= #1.out 17
#19 HUS1_LB01_SFP_MV <= #1.out 18
#20 HUS1_LB01_GT11_MV <= #1.out 19
#21 HUS1_LB01_GT41_MV <= #1.out 20
#22 HUS1_LB01_GT31_MV <= #1.out 21
#23 HUS1_LB01_GT81_MV <= #1.out 22
#24 HUS1_LB01_VVX01_VVX <= #1.out 23
#25 HUS1_LB01_SV21_R <= #1.out 24
#26 KOMFEL_DELAY:fbDelayedAlarmMinutes(_bLarm: #1.out 1, _iMinutes: HUS1_LB01_LC_FL)
#27 HUS1_LB01_LC <= #26.bDelayedAlarm
_END_CFC_
END_PROGRAM

(* POU xEgna Funktionsblock/Modbus/SWEGON GOLD/fbSwegonGOLD_v1, ST *)
FUNCTION_BLOCK fbSwegonGOLD_v1
VAR
	MB_ReadHoldingReg		:FB_MBReadRegs;
	MB_WriteHoldinReg		:FB_MBWriteRegs;
	MB_ReadInputReg		:FB_MBReadInputRegs;
	MB_ReadCoil				:FB_MBReadCoils;
	MB_WriteCoil				:FB_MBWriteCoils;
	MB_InputStatus			:FB_MBReadInputs;

	stGOLD					:ST_SwegonGold_v1;					(* Swegon GOLD-struct *)
	uiSlaveId					:BYTE:=16#FF;						(* Modbus slavadress *)
	iDx							:INT:= 0;								(* Index för sekvensen *)

(*Skrivvariabler*)
	wQuantityRegs				:WORD;
	wWriteMbAdrRegs			:WORD;   							(* Adress att skriva till *)
	wWriteDataRegs				:WORD;							(* Data att skriva till slaven *)

(*Minnesvariabler*)
	rGT11_BV_temp						:REAL;
	rGT11_MIN_temp						:REAL;
	rGT11_MAX_temp					:REAL;
	rGT41_BV_temp						:REAL;
	rGP11_BV_HIGH_temp				:REAL;
	rGP12_BV_HIGH_temp				:REAL;
	rGP11_BV_LOW_temp				:REAL;
	rGP12_BV_LOW_temp				:REAL;

(*Läsdata*)
	iGT81_FrysskydsstempREAD		:INT;
	iDriftlageREAD						:INT;
	iInputStatus1							:INT;						(* iInputStatus1.0 = Operation Active. iInputStatus1.12 = Summalarm A.  iInputStatus1.13 = Summalarm B *)
	iInputStatus2							:INT;						(* iInputStatus2.0 = Re-Heat output. *)


END_VAR
VAR_INPUT
	bEnable								:BOOL;					(* Start läsning *)
	bEnableWrite							:BOOL;					(* Aktivera skrivning *)
	sIPAddr								:STRING(15);				(* IP-adress *)

END_VAR

VAR_IN_OUT
	rGT11_BV								:REAL;						(*Börvärde GT11, tilluftstemperatur*)
	rGT11_MIN							:REAL;						(*Börvärde MIN GT11, tilluftstemperatur*)
	rGT11_MAX							:REAL;						(*Börvärde MAX GT11, tilluftstemperatur*)
	rGT41_BV								:REAL;						(*Börvärde frånluftstemp*)
	rGP11_BV_HIGH						:REAL;						(*Börvärde GP11, tilluftstryck högfart*)
	rGP11_BV_LOW						:REAL;						(*Börvärde GP11, tilluftstryck lågfart*)
	rGP12_BV_HIGH						:REAL;						(*Börvärde GP12, frånluftstryck högfart*)
	rGP12_BV_LOW						:REAL;						(*Börvärde GP12, frånluftstryck lågfart*)

END_VAR

VAR_OUTPUT
	bError:									BOOL;						(*Vi har ett fel, komfel*)
	bBusy:									BOOL;						(*Arbetar*)

(*Beräknad data till utgång*)
	bAggregat_TILL						:BOOL;
	iDriftlage								:INT;						(* 0=Fan not available1=Alarm stop2=Manual total stop (on hand terminal)3=External total stop (digital input)4=Communication total stop5=Communication normal stop6=Communication extended normal stop7=Time channel total stop8=Time channel normal stop9=Time channel extended normal stop10=Low speed=normal stop11=SA Fan starting up12=Fan regulation blocked13=ReCO2 100% recirculation(1.11)14=Morning boost stop(1.11)15=Intermittent night heat stop(1.11)16=After cooling electric heater17=COOL DX switch off delay18=Damper switch off delay19=Manual low speed (on hand terminal)20=External low speed (digital input)21=Extended external low speed22=Communication low speed23=Time channel low speed24=Morning boost low speed25=Intermittent night heat low speed26=Manual high speed (on hand terminal)27=External high speed (digital input)28=Extended external high speed29=Communication high speed30=Time channel high speed31=Summer night cooling high speed32=Filter calibration33=RHX Defrost calibration 34=ReCO2 calibration35=AHU start up36=Re-heat ramp down37=HX ramp down38=Air adjustment39=Fans in operation with active fire alarm40=PX bypass damper adjustment(1.12) *)
	bSummalarmA							:BOOL;
	bSummalarmB							:BOOL;
	bPV01_IND							:BOOL;					(*Driftindikering cirkulationspump*)
	rGP11_MV								:REAL;
	rGP12_MV								:REAL;
	rGF41_MV								:REAL;
	rGF42_MV								:REAL;
	rGP61_MV								:REAL;
	rGP61_limit							:REAL;
	rGP62_MV								:REAL;
	rGP62_limit							:REAL;
	rTF01_level							:REAL;
	rFF01_level							:REAL;
	rSFP									:REAL;
	rGT11_MV								:REAL;
	rGT41_MV								:REAL;
	rGT31_MV								:REAL;
	rGT81_Frysskydsstemp				:REAL;
	rVVX_level							:REAL;
	rSV21_level							:REAL;

END_VAR
CASE iDx OF

0:(*Vänta på start*)
IF bEnable THEN
		bBusy:=TRUE;
		iDx := 5;
ELSE
		bBusy:=FALSE;
		bError:=FALSE;
END_IF


5:(*Läs INPUT registers. Modbus funktion 3*)
	MB_ReadInputReg(
					sIPAddr:= sIPAddr,
					nTCPPort:=502,
					nUnitID:= uiSlaveId ,
					nQuantity:= 35,
					nMBAddr:= 3 ,
					cbLength:= SIZEOF(stGOLD.InputRegs1) ,
					pDestAddr:= ADR(stGOLD.InputRegs1) ,
					bExecute:= TRUE ,
					TTimeout:= T#2s ,
					bBUSY=> ,
					bError=> ,
					nErrId=> ,
					cbRead=> );

	IF NOT MB_ReadInputReg.bBusy AND NOT MB_ReadInputReg.bError THEN
		MB_ReadInputReg(bExecute:=FALSE);
		bError := FALSE;
		bBusy:=FALSE;
		iDx := 10;

	ELSIF MB_ReadInputReg.bError THEN
		MB_ReadInputReg(bExecute:=FALSE);
		iDx := 999;
	END_IF


10:(*Läs INPUT registers. Modbus funktion 3*)
	MB_ReadInputReg(
					sIPAddr:= sIPAddr,
					nTCPPort:=502,
					nUnitID:= uiSlaveId ,
					nQuantity:= 18,
					nMBAddr:= 62 ,
					cbLength:= SIZEOF(stGOLD.InputRegs2) ,
					pDestAddr:= ADR(stGOLD.InputRegs2) ,
					bExecute:= TRUE ,
					TTimeout:= T#2s ,
					bBUSY=> ,
					bError=> ,
					nErrId=> ,
					cbRead=> );

	IF NOT MB_ReadInputReg.bBusy AND NOT MB_ReadInputReg.bError THEN
		MB_ReadInputReg(bExecute:=FALSE);
		bError := FALSE;
		bBusy:=FALSE;
		iDx := 15;

	ELSIF MB_ReadInputReg.bError THEN
		MB_ReadInputReg(bExecute:=FALSE);
		iDx := 999;
	END_IF


15:(*Läs INPUT registers. Modbus funktion 3*)
	MB_ReadInputReg(
					sIPAddr:= sIPAddr,
					nTCPPort:=502,
					nUnitID:= uiSlaveId ,
					nQuantity:= 5,
					nMBAddr:= 90 ,
					cbLength:= SIZEOF(stGOLD.InputRegs3) ,
					pDestAddr:= ADR(stGOLD.InputRegs3) ,
					bExecute:= TRUE ,
					TTimeout:= T#2s ,
					bBUSY=> ,
					bError=> ,
					nErrId=> ,
					cbRead=> );

	IF NOT MB_ReadInputReg.bBusy AND NOT MB_ReadInputReg.bError THEN
		MB_ReadInputReg(bExecute:=FALSE);
		bError := FALSE;
		bBusy:=FALSE;
		iDx := 20;

	ELSIF MB_ReadInputReg.bError THEN
		MB_ReadInputReg(bExecute:=FALSE);
		iDx := 999;
	END_IF


20:(*Läs INPUT registers. Modbus funktion 3*)
	MB_ReadInputReg(
					sIPAddr:= sIPAddr,
					nTCPPort:=502,
					nUnitID:= uiSlaveId ,
					nQuantity:= 1,
					nMBAddr:= 152 ,
					cbLength:= SIZEOF(iGT81_FrysskydsstempREAD) ,
					pDestAddr:= ADR(iGT81_FrysskydsstempREAD) ,
					bExecute:= TRUE ,
					TTimeout:= T#2s ,
					bBUSY=> ,
					bError=> ,
					nErrId=> ,
					cbRead=> );

	IF NOT MB_ReadInputReg.bBusy AND NOT MB_ReadInputReg.bError THEN
		MB_ReadInputReg(bExecute:=FALSE);
		bError := FALSE;
		bBusy:=FALSE;
		iDx := 25;

	ELSIF MB_ReadInputReg.bError THEN
		MB_ReadInputReg(bExecute:=FALSE);
		iDx := 999;
	END_IF


25:(*Läs INPUT registers. Modbus funktion 3*)
	MB_ReadInputReg(
					sIPAddr:= sIPAddr,
					nTCPPort:=502,
					nUnitID:= uiSlaveId ,
					nQuantity:= 1,
					nMBAddr:= 591 ,
					cbLength:= SIZEOF(iDriftlageREAD) ,
					pDestAddr:= ADR(iDriftlageREAD) ,
					bExecute:= TRUE ,
					TTimeout:= T#2s ,
					bBUSY=> ,
					bError=> ,
					nErrId=> ,
					cbRead=> );

	IF NOT MB_ReadInputReg.bBusy AND NOT MB_ReadInputReg.bError THEN
		MB_ReadInputReg(bExecute:=FALSE);
		bError := FALSE;
		bBusy:=FALSE;
		iDx := 30;

	ELSIF MB_ReadInputReg.bError THEN
		MB_ReadInputReg(bExecute:=FALSE);
		iDx := 999;
	END_IF


30:(*Läs HOLDING registers. Modbus funktion 4*)
	MB_ReadHoldingReg(
					sIPAddr:= sIPAddr,
					nTCPPort:=502,
					nUnitID:= uiSlaveId ,
					nQuantity:= 4,
					nMBAddr:= 18 ,
					cbLength:= SIZEOF(stGOLD.HoldingRegs1) ,
					pDestAddr:= ADR(stGOLD.HoldingRegs1) ,
					bExecute:= TRUE ,
					TTimeout:= T#2s ,
					bBUSY=> ,
					bError=> ,
					nErrId=> ,
					cbRead=> );

	IF NOT MB_ReadHoldingReg.bBusy AND NOT MB_ReadHoldingReg.bError THEN
		MB_ReadHoldingReg(bExecute:=FALSE);
		bError := FALSE;
		bBusy:=FALSE;
		iDx := 35;

	ELSIF MB_ReadInputReg.bError THEN
		MB_ReadHoldingReg(bExecute:=FALSE);
		iDx := 999;
	END_IF


35:(*Läs HOLDING registers. Modbus funktion 4*)
	MB_ReadHoldingReg(
					sIPAddr:= sIPAddr,
					nTCPPort:=502,
					nUnitID:= uiSlaveId ,
					nQuantity:= 6,
					nMBAddr:= 131 ,
					cbLength:= SIZEOF(stGOLD.HoldingRegs2) ,
					pDestAddr:= ADR(stGOLD.HoldingRegs2) ,
					bExecute:= TRUE ,
					TTimeout:= T#2s ,
					bBUSY=> ,
					bError=> ,
					nErrId=> ,
					cbRead=> );

	IF NOT MB_ReadHoldingReg.bBusy AND NOT MB_ReadHoldingReg.bError THEN
		MB_ReadHoldingReg(bExecute:=FALSE);
		bError := FALSE;
		bBusy:=FALSE;
		iDx := 40;

	ELSIF MB_ReadHoldingReg.bError THEN
		MB_ReadHoldingReg(bExecute:=FALSE);
		iDx := 999;
	END_IF


40:(*Läs INPUT status*)
	MB_InputStatus(
					sIPAddr:= sIPAddr,
					nTCPPort:=502,
					nUnitID:= uiSlaveId ,
					nQuantity:= 16,
					nMBAddr:= 0 ,
					cbLength:= SIZEOF(iInputStatus1) ,
					pDestAddr:= ADR(iInputStatus1) ,
					bExecute:= TRUE ,
					TTimeout:= T#2s ,
					bBUSY=> ,
					bError=> ,
					nErrId=> ,
					cbRead=> );

	IF NOT MB_InputStatus.bBusy AND NOT MB_InputStatus.bError THEN
		MB_InputStatus(bExecute:=FALSE);
		bError := FALSE;
		bBusy:=FALSE;
		iDx := 45;

	ELSIF MB_InputStatus.bError THEN
		MB_InputStatus(bExecute:=FALSE);
		iDx := 999;
	END_IF


45:(*Läs INPUT status*)
	MB_InputStatus(
					sIPAddr:= sIPAddr,
					nTCPPort:=502,
					nUnitID:= uiSlaveId ,
					nQuantity:= 3,
					nMBAddr:= 37,
					cbLength:= SIZEOF(iInputStatus2) ,
					pDestAddr:= ADR(iInputStatus2) ,
					bExecute:= TRUE ,
					TTimeout:= T#2s ,
					bBUSY=> ,
					bError=> ,
					nErrId=> ,
					cbRead=> );

	IF NOT MB_InputStatus.bBusy AND NOT MB_InputStatus.bError THEN
		MB_InputStatus(bExecute:=FALSE);
		bError := FALSE;
		bBusy:=FALSE;
		iDx := 95;

	ELSIF MB_InputStatus.bError THEN
		MB_InputStatus(bExecute:=FALSE);
		iDx := 999;
	END_IF

(*Anropa action och beräkna läst data*)
95:
	actCalculateData;

(*Anropa actions och kontrollera om skrivning behövs*)
105:
	fbSwegonGOLD_v1.actCheckWrite4x0019;
110:
	fbSwegonGOLD_v1.actCheckWrite4x0020;
115:
	fbSwegonGOLD_v1.actCheckWrite4x0021;
120:
	fbSwegonGOLD_v1.actCheckWrite4x0022;
125:
	fbSwegonGOLD_v1.actCheckWrite4x0132;
130:
	fbSwegonGOLD_v1.actCheckWrite4x0135;
135:
	fbSwegonGOLD_v1.actCheckWrite4x0136;
140:
	fbSwegonGOLD_v1.actCheckWrite4x0137;


200:	(*Skriv data*)
MB_WriteHoldinReg(
				sIPAddr:= sIPAddr,
				nTCPPort:=502,
				nUnitID:= uiSlaveId ,
				nQuantity:= wQuantityRegs,
				nMBAddr:= wWriteMbAdrRegs ,
				cbLength:= SIZEOF(wWriteDataRegs) ,
				pSrcAddr:= ADR(wWriteDataRegs) ,
				bExecute:= TRUE ,
				TTimeout:= T#2s ,
				bBUSY=> ,
				bError=> ,
				nErrId=> );

	IF NOT MB_WriteHoldinReg.bBusy AND NOT MB_WriteHoldinReg.bError THEN
		MB_WriteHoldinReg(bExecute:=FALSE);
		bError := FALSE;
		bBusy:=FALSE;
		iDx := 0;

	ELSIF MB_WriteHoldinReg.bError THEN
		MB_WriteHoldinReg(bExecute:=FALSE);
		iDx := 999;
	END_IF


999: (* Error *)
	bError := TRUE;
	MB_ReadHoldingReg(bExecute:=FALSE);
	MB_WriteHoldinReg(bExecute:=FALSE);
	MB_ReadInputReg(bExecute:=FALSE);
	MB_ReadCoil(bExecute:=FALSE);
	MB_WriteCoil(bExecute:=FALSE);
	MB_InputStatus(bExecute:=FALSE);

	bBusy:=FALSE;
	iDx := 0;


END_CASE
END_FUNCTION_BLOCK
ACTION actCalculateData:
(*Beräkning/konvertering av signaler till utgång*)


(* MÄTVÄRDEN & UTSIGNALER *)

	rGP11_MV:=						INT_TO_REAL(stGOLD.InputRegs1.SA_Duct_pressure)/10;							(*3x0008*)
	rGP12_MV:=						INT_TO_REAL(stGOLD.InputRegs1.EA_Duct_pressure)/10;							(*3x0010*)
	rGF41_MV:=						INT_TO_REAL(stGOLD.InputRegs1.SA_Air_Flow);									(*3x0004*)
	rGF42_MV:=						INT_TO_REAL(stGOLD.InputRegs1.EA_Air_Flow);									(*3x0006*)
	rGP61_MV:=						INT_TO_REAL(stGOLD.InputRegs1.SA_AHU_filter_pressure_level)/10;				(*3x0027*)
	rGP61_limit:=						INT_TO_REAL(stGOLD.InputRegs1.SA_AHU_filter_pressure_alarm_limit)/10;		(*3x0028*)
	rGP62_MV:=						INT_TO_REAL(stGOLD.InputRegs1.EA_AHU_filter_pressure_level)/10;				(*3x0029*)
	rGP62_limit:=						INT_TO_REAL(stGOLD.InputRegs1.EA_AHU_filter_pressure_alarm_limit)/10;		(*3x0030*)
	rTF01_level:=						INT_TO_REAL(stGOLD.InputRegs1.SA_Fan_level)/100;								(*3x0037*)
	rFF01_level:=						INT_TO_REAL(stGOLD.InputRegs1.EA_Fan_level)/100;								(*3x0038*)

	rSFP:=								INT_TO_REAL(stGOLD.InputRegs2.SFP)/100;											(*3x0063*)
	rGT11_MV:=						INT_TO_REAL(stGOLD.InputRegs2.SA_Temperature)/100;								(*3x0064*)
	rGT41_MV:=						INT_TO_REAL(stGOLD.InputRegs2.EA_Temperature_PXCX)/100;						(*3x0069*)
	rGT31_MV:=						INT_TO_REAL(stGOLD.InputRegs2.Outdoor_temperature)/100;						(*3x0073*)

	rVVX_level:=						INT_TO_REAL(stGOLD.InputRegs3.Heat_exchanger_regulator_level)/100;			(*3x0091*)
	rSV21_level:=						INT_TO_REAL(stGOLD.InputRegs3.Reheat_output_level)/100;						(*3x0095*)

	rGT81_Frysskydsstemp:=			INT_TO_REAL(iGT81_FrysskydsstempREAD)/100;										(*3x0153*)
	iDriftlage:=							iDriftlageREAD;																			(*3x0592*)			(* 0=Fan not available1=Alarm stop2=Manual total stop (on hand terminal)3=External total stop (digital input)4=Communication total stop5=Communication normal stop6=Communication extended normal stop7=Time channel total stop8=Time channel normal stop9=Time channel extended normal stop10=Low speed=normal stop11=SA Fan starting up12=Fan regulation blocked13=ReCO2 100% recirculation(1.11)14=Morning boost stop(1.11)15=Intermittent night heat stop(1.11)16=After cooling electric heater17=COOL DX switch off delay18=Damper switch off delay19=Manual low speed (on hand terminal)20=External low speed (digital input)21=Extended external low speed22=Communication low speed23=Time channel low speed24=Morning boost low speed25=Intermittent night heat low speed26=Manual high speed (on hand terminal)27=External high speed (digital input)28=Extended external high speed29=Communication high speed30=Time channel high speed31=Summer night cooling high speed32=Filter calibration33=RHX Defrost calibration 34=ReCO2 calibration35=AHU start up36=Re-heat ramp down37=HX ramp down38=Air adjustment39=Fans in operation with active fire alarm40=PX bypass damper adjustment(1.12) *)




(* INIDKERINGAR & LARM *)
	bAggregat_TILL:=				iInputStatus1.0;																			(*1x0001*)
	bSummalarmA:=					iInputStatus1.12;																			(*1x0013*)
	bSummalarmB:=					iInputStatus1.13;																			(*1x0014*)
	bPV01_IND:=						iInputStatus2.0;																			(*1x0038*)



(* GÅ TILL NÄSTA STEG *)
	iDx := 105;
END_ACTION
ACTION actCheckWrite4x0019:
(* Kolla om vi skall skriva till 4x0019 *)

IF
	stGOLD.HoldingRegs1.SA_low_speed_pressure_setpoint<>REAL_TO_INT(rGP11_BV_LOW_temp*10)

THEN
	rGP11_BV_LOW_temp:=INT_TO_REAL(stGOLD.HoldingRegs1.SA_low_speed_pressure_setpoint)/10;
	rGP11_BV_LOW:=INT_TO_REAL(stGOLD.HoldingRegs1.SA_low_speed_pressure_setpoint)/10;

	iDx:=110;     (*110*)
ELSIF
	bEnableWrite AND bError=FALSE AND
	rGP11_BV_LOW<> rGP11_BV_LOW_temp

THEN
	rGP11_BV_LOW_temp:=rGP11_BV_LOW;

	wQuantityRegs:=1;
	wWriteMbAdrRegs:=18;
	wWriteDataRegs:= REAL_TO_INT(rGP11_BV_LOW*10);

	iDx := 200;

ELSE
	iDx:=110;  (*110*)
END_IF
END_ACTION
ACTION actCheckWrite4x0020:
(* Kolla om vi skall skriva till 4x0020 *)

IF
	stGOLD.HoldingRegs1.EA_low_speed_pressure_setpoint<>REAL_TO_INT(rGP12_BV_LOW_temp*10)

THEN
	rGP12_BV_LOW_temp:=INT_TO_REAL(stGOLD.HoldingRegs1.EA_low_speed_pressure_setpoint)/10;
	rGP12_BV_LOW:=INT_TO_REAL(stGOLD.HoldingRegs1.EA_low_speed_pressure_setpoint)/10;

	iDx:=115;  (*115*)
ELSIF
	bEnableWrite AND bError=FALSE AND
	rGP12_BV_LOW<> rGP12_BV_LOW_temp

THEN
	rGP12_BV_LOW_temp:=rGP12_BV_LOW;

	wQuantityRegs:=1;
	wWriteMbAdrRegs:=19;
	wWriteDataRegs:= REAL_TO_INT(rGP12_BV_LOW*10);

	iDx := 200;

ELSE
	iDx:=115;
END_IF
END_ACTION
ACTION actCheckWrite4x0021:
(* Kolla om vi skall skriva till 4x0021 *)

IF
	stGOLD.HoldingRegs1.SA_high_speed_pressure_setpoint<>REAL_TO_INT(rGP11_BV_HIGH_temp*10)

THEN
	rGP11_BV_HIGH_temp:=INT_TO_REAL(stGOLD.HoldingRegs1.SA_high_speed_pressure_setpoint)/10;
	rGP11_BV_HIGH:=INT_TO_REAL(stGOLD.HoldingRegs1.SA_high_speed_pressure_setpoint)/10;

	iDx:=120;  (*120*)
ELSIF
	bEnableWrite AND bError=FALSE AND
	rGP11_BV_HIGH<> rGP11_BV_HIGH_temp

THEN
	rGP11_BV_HIGH_temp:=rGP11_BV_HIGH;

	wQuantityRegs:=1;
	wWriteMbAdrRegs:=20;
	wWriteDataRegs:= REAL_TO_INT(rGP11_BV_HIGH*10);

	iDx := 200;

ELSE
	iDx:=120;
END_IF
END_ACTION
ACTION actCheckWrite4x0022:
(* Kolla om vi skall skriva till 4x0022 *)

IF
	stGOLD.HoldingRegs1.EA_high_speed_pressure_setpoint<>REAL_TO_INT(rGP12_BV_HIGH_temp*10)

THEN
	rGP12_BV_HIGH_temp:=INT_TO_REAL(stGOLD.HoldingRegs1.EA_high_speed_pressure_setpoint)/10;
	rGP12_BV_HIGH:=INT_TO_REAL(stGOLD.HoldingRegs1.EA_high_speed_pressure_setpoint)/10;

	iDx:=125;  (*125*)
ELSIF
	bEnableWrite AND bError=FALSE AND
	rGP12_BV_HIGH<> rGP12_BV_HIGH_temp

THEN
	rGP12_BV_HIGH_temp:=rGP12_BV_HIGH;

	wQuantityRegs:=1;
	wWriteMbAdrRegs:=21;
	wWriteDataRegs:= REAL_TO_INT(rGP12_BV_HIGH*10);

	iDx := 200;

ELSE
	iDx:=125;
END_IF
END_ACTION
ACTION actCheckWrite4x0132:
(* Kolla om vi skall skriva till 4x0132 *)

IF
	stGOLD.HoldingRegs2.SA_temperature_setpoint<>REAL_TO_INT(rGT11_BV_temp*100)

THEN
	rGT11_BV_temp:=INT_TO_REAL(stGOLD.HoldingRegs2.SA_temperature_setpoint)/100;
	rGT11_BV:=INT_TO_REAL(stGOLD.HoldingRegs2.SA_temperature_setpoint)/100;

	iDx:=130;
ELSIF
	bEnableWrite AND bError=FALSE AND
	rGT11_BV<> rGT11_BV_temp

THEN
	rGT11_BV_temp:=rGT11_BV;

	wQuantityRegs:=1;
	wWriteMbAdrRegs:=131;
	wWriteDataRegs:= REAL_TO_INT(rGT11_BV*100);

	iDx := 200;

ELSE
	iDx:=130;
END_IF
END_ACTION
ACTION actCheckWrite4x0135:
(* Kolla om vi skall skriva till 4x0135 *)

IF
	stGOLD.HoldingRegs2.EA_Room_temperature_setpoint<>REAL_TO_INT(rGT41_BV_temp*100)

THEN
	rGT41_BV_temp:=INT_TO_REAL(stGOLD.HoldingRegs2.EA_Room_temperature_setpoint)/100;
	rGT41_BV:=INT_TO_REAL(stGOLD.HoldingRegs2.EA_Room_temperature_setpoint)/100;

	iDx:=135;
ELSIF
	bEnableWrite AND bError=FALSE AND
	rGT41_BV<> rGT41_BV_temp

THEN
	rGT41_BV_temp:=rGT41_BV;

	wQuantityRegs:=1;
	wWriteMbAdrRegs:=134;
	wWriteDataRegs:= REAL_TO_INT(rGT41_BV*100);

	iDx := 200;

ELSE
	iDx:=135;
END_IF
END_ACTION
ACTION actCheckWrite4x0136:
(* Kolla om vi skall skriva till 4x0136 *)

IF
	stGOLD.HoldingRegs2.SA_min_temp_setpoint<>REAL_TO_INT(rGT11_MIN_temp*100)

THEN
	rGT11_MIN_temp:=INT_TO_REAL(stGOLD.HoldingRegs2.SA_min_temp_setpoint)/100;
	rGT11_MIN:=INT_TO_REAL(stGOLD.HoldingRegs2.SA_min_temp_setpoint)/100;

	iDx:=140;
ELSIF
	bEnableWrite AND bError=FALSE AND
	rGT11_MIN<> rGT11_MIN_temp

THEN
	rGT11_MIN_temp:=rGT11_MIN;

	wQuantityRegs:=1;
	wWriteMbAdrRegs:=135;
	wWriteDataRegs:= REAL_TO_INT(rGT11_MIN*100);

	iDx := 200;

ELSE
	iDx:=140;
END_IF
END_ACTION
ACTION actCheckWrite4x0137:
(* Kolla om vi skall skriva till 4x0137 *)

IF
	stGOLD.HoldingRegs2.SA_max_temp_setpoint<>REAL_TO_INT(rGT11_MAX_temp*100)

THEN
	rGT11_MAX_temp:=INT_TO_REAL(stGOLD.HoldingRegs2.SA_max_temp_setpoint)/100;
	rGT11_MAX:=INT_TO_REAL(stGOLD.HoldingRegs2.SA_max_temp_setpoint)/100;

	iDx:=0;
ELSIF
	bEnableWrite AND bError=FALSE AND
	rGT11_MAX<> rGT11_MAX_temp

THEN
	rGT11_MAX_temp:=rGT11_MAX;

	wQuantityRegs:=1;
	wWriteMbAdrRegs:=136;
	wWriteDataRegs:= REAL_TO_INT(rGT11_MAX*100);

	iDx := 200;

ELSE
	iDx:=0;
END_IF
END_ACTION

(* POU SYSTEM/_Modbus TCP/GOLD_AGGREGAT/MODBUS_LB02, CFC *)
PROGRAM MODBUS_LB02
VAR

	KOMFEL_DELAY: fbDelayedAlarmMinutes;

(*LB02*)
	LB02_MODBUS: fbSwegonGOLD_v1;
	bEnableRead2			:BOOL:=TRUE;
	bEnableWrite2			:BOOL:=TRUE;		(*SÄTT TILL INITIAL TRUE VID DRIFTSÄTTNING*)
	bError2					:BOOL;
	bBusy2					:BOOL;

	rDUMMY_GT11_MIN2	:REAL;
	rDUMMY_GT11_MAX2	:REAL;
	rDUMMY_GT41_BV2		:REAL;
	rDUMMY_GP11_LOW2	:REAL;
	rDUMMY_GP12_LOW2	:REAL;
	bLB02_TILL				:BOOL;


END_VAR
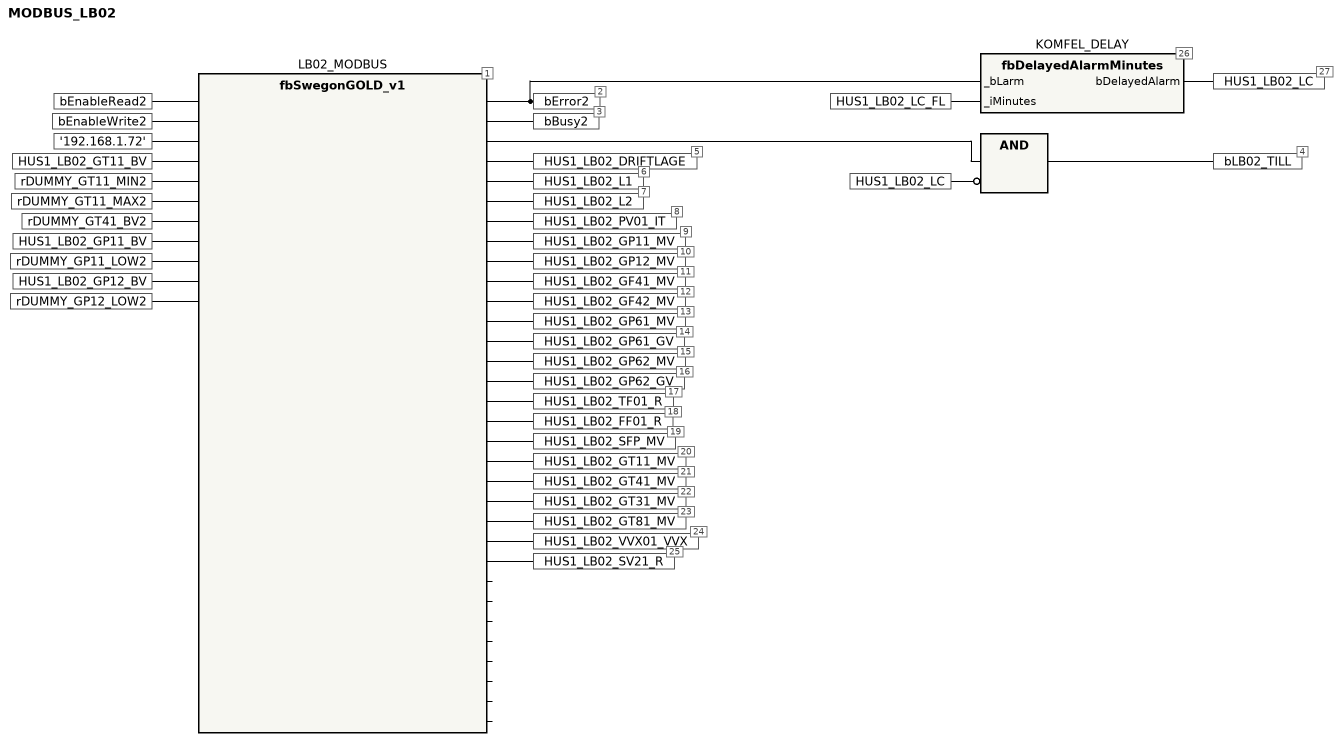
_CFC_ (* Continuous Function Chart, elements in execution order *)
#0 AND(#1.out 3, NOT HUS1_LB02_LC)
#1 LB02_MODBUS:fbSwegonGOLD_v1(bEnableRead2, bEnableWrite2, '192.168.1.72', HUS1_LB02_GT11_BV, rDUMMY_GT11_MIN2, rDUMMY_GT11_MAX2, rDUMMY_GT41_BV2, HUS1_LB02_GP11_BV, rDUMMY_GP11_LOW2, HUS1_LB02_GP12_BV, rDUMMY_GP12_LOW2)
#2 bError2 <= #1.out 1
#3 bBusy2 <= #1.out 2
#4 bLB02_TILL <= #0
#5 HUS1_LB02_DRIFTLAGE <= #1.out 4
#6 HUS1_LB02_L1 <= #1.out 5
#7 HUS1_LB02_L2 <= #1.out 6
#8 HUS1_LB02_PV01_IT <= #1.out 7
#9 HUS1_LB02_GP11_MV <= #1.out 8
#10 HUS1_LB02_GP12_MV <= #1.out 9
#11 HUS1_LB02_GF41_MV <= #1.out 10
#12 HUS1_LB02_GF42_MV <= #1.out 11
#13 HUS1_LB02_GP61_MV <= #1.out 12
#14 HUS1_LB02_GP61_GV <= #1.out 13
#15 HUS1_LB02_GP62_MV <= #1.out 14
#16 HUS1_LB02_GP62_GV <= #1.out 15
#17 HUS1_LB02_TF01_R <= #1.out 16
#18 HUS1_LB02_FF01_R <= #1.out 17
#19 HUS1_LB02_SFP_MV <= #1.out 18
#20 HUS1_LB02_GT11_MV <= #1.out 19
#21 HUS1_LB02_GT41_MV <= #1.out 20
#22 HUS1_LB02_GT31_MV <= #1.out 21
#23 HUS1_LB02_GT81_MV <= #1.out 22
#24 HUS1_LB02_VVX01_VVX <= #1.out 23
#25 HUS1_LB02_SV21_R <= #1.out 24
#26 KOMFEL_DELAY:fbDelayedAlarmMinutes(_bLarm: #1.out 1, _iMinutes: HUS1_LB02_LC_FL)
#27 HUS1_LB02_LC <= #26.bDelayedAlarm
_END_CFC_
END_PROGRAM

(* POU SYSTEM/_Modbus TCP/GOLD_AGGREGAT/MODBUS_LB03, CFC *)
PROGRAM MODBUS_LB03
VAR

	KOMFEL_DELAY: fbDelayedAlarmMinutes;

(*LB03*)
	LB03_MODBUS: fbSwegonGOLD_v1;
	bEnableRead3			:BOOL:=TRUE;
	bEnableWrite3			:BOOL:=TRUE;				(*SÄTT TILL INITIAL TRUE VID DRIFTSÄTTNING*)
	bError3					:BOOL;
	bBusy3					:BOOL;

	rDUMMY_GT11_MIN3	:REAL;
	rDUMMY_GT11_MAX3	:REAL;
	rDUMMY_GT41_BV3		:REAL;
	rDUMMY_GP11_LOW3	:REAL;
	rDUMMY_GP12_LOW3	:REAL;
	bLB03_TILL				:BOOL;

END_VAR
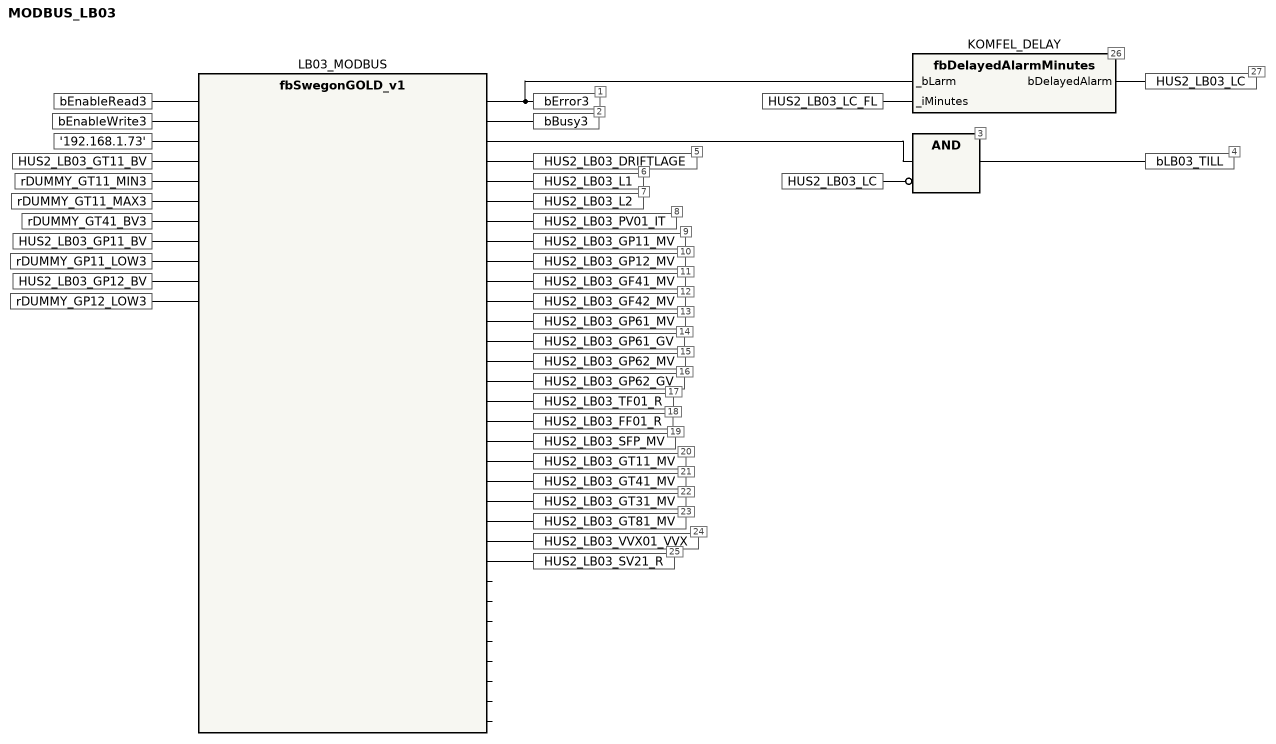
_CFC_ (* Continuous Function Chart, elements in execution order *)
#0 LB03_MODBUS:fbSwegonGOLD_v1(bEnableRead3, bEnableWrite3, '192.168.1.73', HUS2_LB03_GT11_BV, rDUMMY_GT11_MIN3, rDUMMY_GT11_MAX3, rDUMMY_GT41_BV3, HUS2_LB03_GP11_BV, rDUMMY_GP11_LOW3, HUS2_LB03_GP12_BV, rDUMMY_GP12_LOW3)
#1 bError3 <= #0.out 1
#2 bBusy3 <= #0.out 2
#3 AND(#0.out 3, NOT HUS2_LB03_LC)
#4 bLB03_TILL <= #3
#5 HUS2_LB03_DRIFTLAGE <= #0.out 4
#6 HUS2_LB03_L1 <= #0.out 5
#7 HUS2_LB03_L2 <= #0.out 6
#8 HUS2_LB03_PV01_IT <= #0.out 7
#9 HUS2_LB03_GP11_MV <= #0.out 8
#10 HUS2_LB03_GP12_MV <= #0.out 9
#11 HUS2_LB03_GF41_MV <= #0.out 10
#12 HUS2_LB03_GF42_MV <= #0.out 11
#13 HUS2_LB03_GP61_MV <= #0.out 12
#14 HUS2_LB03_GP61_GV <= #0.out 13
#15 HUS2_LB03_GP62_MV <= #0.out 14
#16 HUS2_LB03_GP62_GV <= #0.out 15
#17 HUS2_LB03_TF01_R <= #0.out 16
#18 HUS2_LB03_FF01_R <= #0.out 17
#19 HUS2_LB03_SFP_MV <= #0.out 18
#20 HUS2_LB03_GT11_MV <= #0.out 19
#21 HUS2_LB03_GT41_MV <= #0.out 20
#22 HUS2_LB03_GT31_MV <= #0.out 21
#23 HUS2_LB03_GT81_MV <= #0.out 22
#24 HUS2_LB03_VVX01_VVX <= #0.out 23
#25 HUS2_LB03_SV21_R <= #0.out 24
#26 KOMFEL_DELAY:fbDelayedAlarmMinutes(_bLarm: #0.out 1, _iMinutes: HUS2_LB03_LC_FL)
#27 HUS2_LB03_LC <= #26.bDelayedAlarm
_END_CFC_
END_PROGRAM

(* POU SYSTEM/_Modbus TCP/GOLD_AGGREGAT/MODBUS_LB04, CFC *)
PROGRAM MODBUS_LB04
VAR

	KOMFEL_DELAY: fbDelayedAlarmMinutes;

(*LB04*)
	LB04_MODBUS: fbSwegonGOLD_v1;
	bEnableRead4			:BOOL:=TRUE;
	bEnableWrite4			:BOOL:=TRUE;			(*SÄTT TILL INITIAL TRUE VID DRIFTSÄTTNING*)
	bError4					:BOOL;
	bBusy4					:BOOL;

	rDUMMY_GT11_MIN4	:REAL;
	rDUMMY_GT11_MAX4	:REAL;
	rDUMMY_GT41_BV4		:REAL;
	rDUMMY_GP11_LOW4	:REAL;
	rDUMMY_GP12_LOW4	:REAL;
	bLB04_TILL				:BOOL;



END_VAR
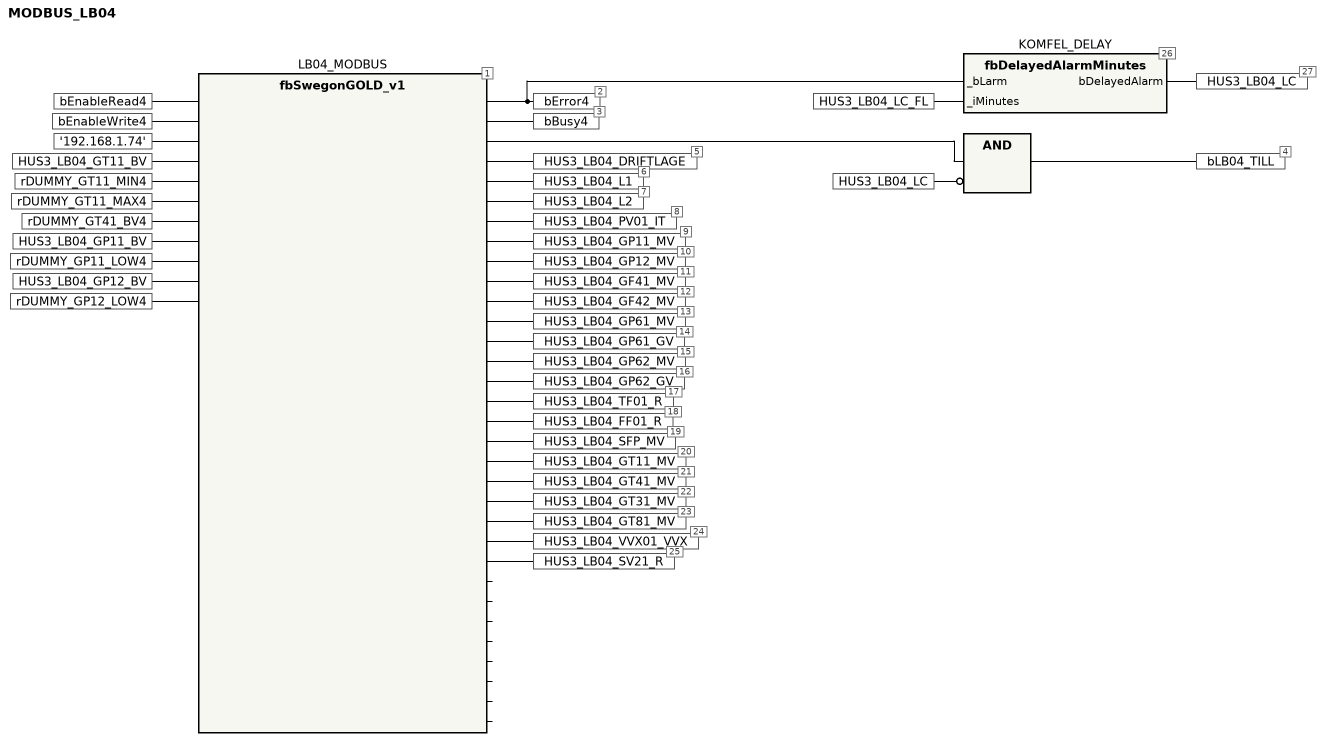
_CFC_ (* Continuous Function Chart, elements in execution order *)
#0 AND(#1.out 3, NOT HUS3_LB04_LC)
#1 LB04_MODBUS:fbSwegonGOLD_v1(bEnableRead4, bEnableWrite4, '192.168.1.74', HUS3_LB04_GT11_BV, rDUMMY_GT11_MIN4, rDUMMY_GT11_MAX4, rDUMMY_GT41_BV4, HUS3_LB04_GP11_BV, rDUMMY_GP11_LOW4, HUS3_LB04_GP12_BV, rDUMMY_GP12_LOW4)
#2 bError4 <= #1.out 1
#3 bBusy4 <= #1.out 2
#4 bLB04_TILL <= #0
#5 HUS3_LB04_DRIFTLAGE <= #1.out 4
#6 HUS3_LB04_L1 <= #1.out 5
#7 HUS3_LB04_L2 <= #1.out 6
#8 HUS3_LB04_PV01_IT <= #1.out 7
#9 HUS3_LB04_GP11_MV <= #1.out 8
#10 HUS3_LB04_GP12_MV <= #1.out 9
#11 HUS3_LB04_GF41_MV <= #1.out 10
#12 HUS3_LB04_GF42_MV <= #1.out 11
#13 HUS3_LB04_GP61_MV <= #1.out 12
#14 HUS3_LB04_GP61_GV <= #1.out 13
#15 HUS3_LB04_GP62_MV <= #1.out 14
#16 HUS3_LB04_GP62_GV <= #1.out 15
#17 HUS3_LB04_TF01_R <= #1.out 16
#18 HUS3_LB04_FF01_R <= #1.out 17
#19 HUS3_LB04_SFP_MV <= #1.out 18
#20 HUS3_LB04_GT11_MV <= #1.out 19
#21 HUS3_LB04_GT41_MV <= #1.out 20
#22 HUS3_LB04_GT31_MV <= #1.out 21
#23 HUS3_LB04_GT81_MV <= #1.out 22
#24 HUS3_LB04_VVX01_VVX <= #1.out 23
#25 HUS3_LB04_SV21_R <= #1.out 24
#26 KOMFEL_DELAY:fbDelayedAlarmMinutes(_bLarm: #1.out 1, _iMinutes: HUS3_LB04_LC_FL)
#27 HUS3_LB04_LC <= #26.bDelayedAlarm
_END_CFC_
END_PROGRAM

(* POU SYSTEM/_Modbus TCP/GOLD_AGGREGAT/MODBUS_LB05, CFC *)
PROGRAM MODBUS_LB05
VAR

	KOMFEL_DELAY: fbDelayedAlarmMinutes;

(*LB05*)
	LB05_MODBUS: fbSwegonGOLD_v1;
	bEnableRead5			:BOOL:=TRUE;
	bEnableWrite5			:BOOL:=TRUE;				(*SÄTT TILL INITIAL TRUE VID DRIFTSÄTTNING*)
	bError5					:BOOL;
	bBusy5					:BOOL;

	rDUMMY_GT11_MIN5	:REAL;
	rDUMMY_GT11_MAX5	:REAL;
	rDUMMY_GT41_BV5		:REAL;
	rDUMMY_GP11_LOW5	:REAL;
	rDUMMY_GP12_LOW5	:REAL;
	bLB05_TILL				:BOOL;


END_VAR
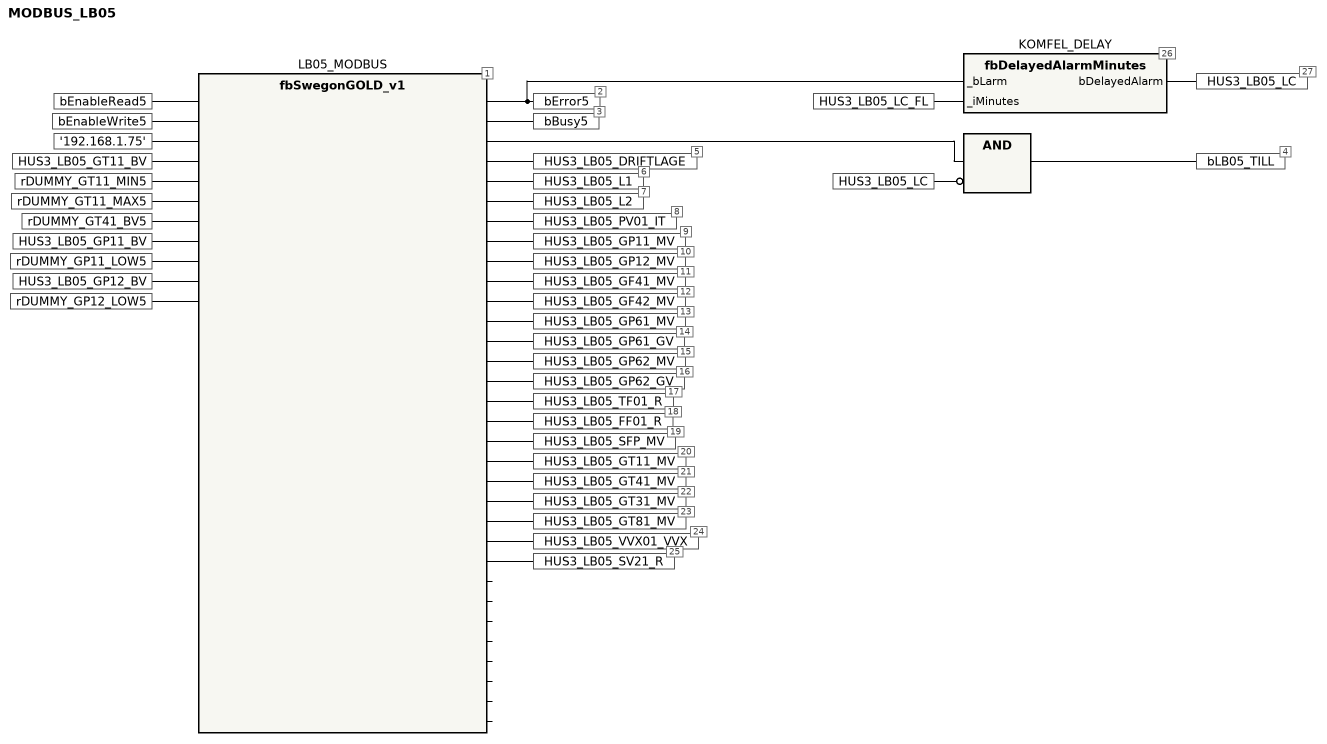
_CFC_ (* Continuous Function Chart, elements in execution order *)
#0 AND(#1.out 3, NOT HUS3_LB05_LC)
#1 LB05_MODBUS:fbSwegonGOLD_v1(bEnableRead5, bEnableWrite5, '192.168.1.75', HUS3_LB05_GT11_BV, rDUMMY_GT11_MIN5, rDUMMY_GT11_MAX5, rDUMMY_GT41_BV5, HUS3_LB05_GP11_BV, rDUMMY_GP11_LOW5, HUS3_LB05_GP12_BV, rDUMMY_GP12_LOW5)
#2 bError5 <= #1.out 1
#3 bBusy5 <= #1.out 2
#4 bLB05_TILL <= #0
#5 HUS3_LB05_DRIFTLAGE <= #1.out 4
#6 HUS3_LB05_L1 <= #1.out 5
#7 HUS3_LB05_L2 <= #1.out 6
#8 HUS3_LB05_PV01_IT <= #1.out 7
#9 HUS3_LB05_GP11_MV <= #1.out 8
#10 HUS3_LB05_GP12_MV <= #1.out 9
#11 HUS3_LB05_GF41_MV <= #1.out 10
#12 HUS3_LB05_GF42_MV <= #1.out 11
#13 HUS3_LB05_GP61_MV <= #1.out 12
#14 HUS3_LB05_GP61_GV <= #1.out 13
#15 HUS3_LB05_GP62_MV <= #1.out 14
#16 HUS3_LB05_GP62_GV <= #1.out 15
#17 HUS3_LB05_TF01_R <= #1.out 16
#18 HUS3_LB05_FF01_R <= #1.out 17
#19 HUS3_LB05_SFP_MV <= #1.out 18
#20 HUS3_LB05_GT11_MV <= #1.out 19
#21 HUS3_LB05_GT41_MV <= #1.out 20
#22 HUS3_LB05_GT31_MV <= #1.out 21
#23 HUS3_LB05_GT81_MV <= #1.out 22
#24 HUS3_LB05_VVX01_VVX <= #1.out 23
#25 HUS3_LB05_SV21_R <= #1.out 24
#26 KOMFEL_DELAY:fbDelayedAlarmMinutes(_bLarm: #1.out 1, _iMinutes: HUS3_LB05_LC_FL)
#27 HUS3_LB05_LC <= #26.bDelayedAlarm
_END_CFC_
END_PROGRAM

(* POU SYSTEM/_Modbus TCP/GOLD_AGGREGAT/MODBUS_LB06, CFC *)
PROGRAM MODBUS_LB06
VAR

	KOMFEL_DELAY: fbDelayedAlarmMinutes;

(*LB06*)
	LB06_MODBUS: fbSwegonGOLD_v1;
	bEnableRead6			:BOOL:=TRUE;
	bEnableWrite6			:BOOL:=TRUE;			(*SÄTT TILL INITIAL TRUE VID DRIFTSÄTTNING*)
	bError6					:BOOL;
	bBusy6					:BOOL;

	rDUMMY_GT11_BV6		:REAL;
	bLB06_TILL				:BOOL;


END_VAR
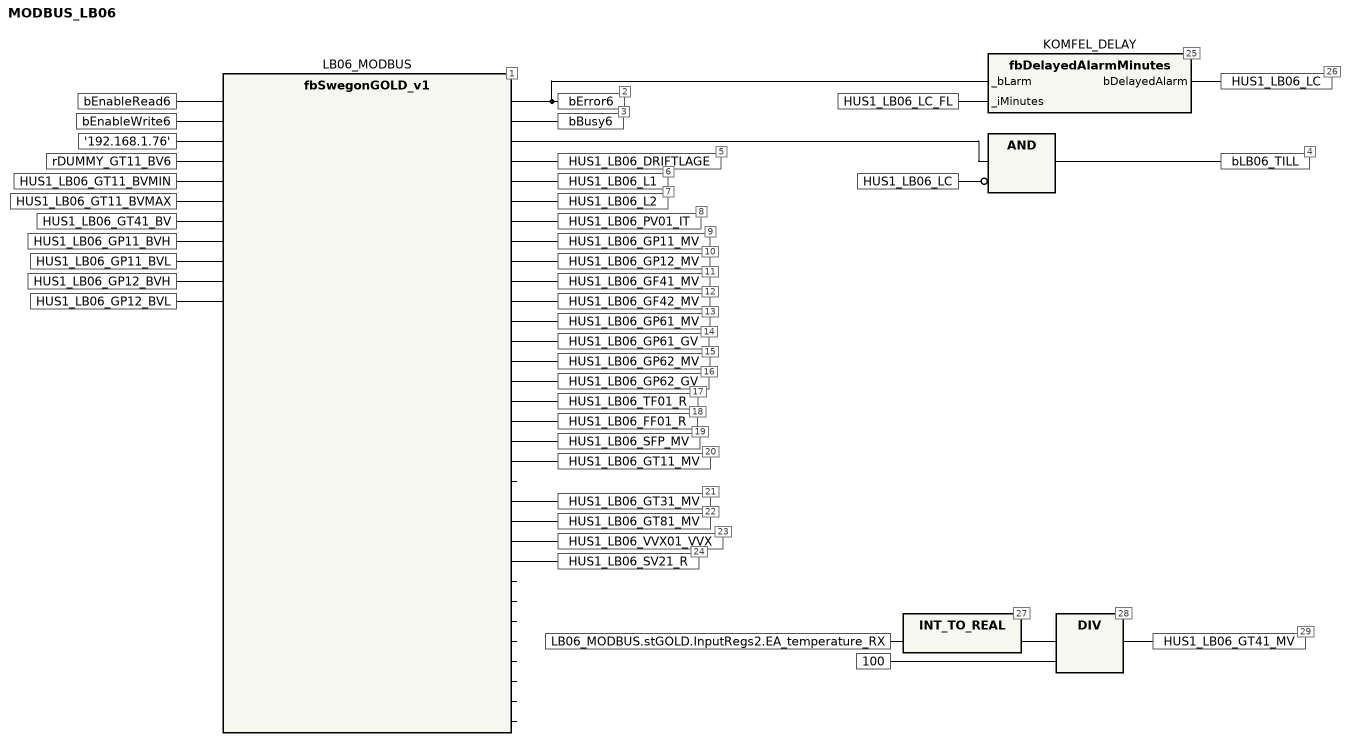
_CFC_ (* Continuous Function Chart, elements in execution order *)
#0 AND(#1.out 3, NOT HUS1_LB06_LC)
#1 LB06_MODBUS:fbSwegonGOLD_v1(bEnableRead6, bEnableWrite6, '192.168.1.76', rDUMMY_GT11_BV6, HUS1_LB06_GT11_BVMIN, HUS1_LB06_GT11_BVMAX, HUS1_LB06_GT41_BV, HUS1_LB06_GP11_BVH, HUS1_LB06_GP11_BVL, HUS1_LB06_GP12_BVH, HUS1_LB06_GP12_BVL)
#2 bError6 <= #1.out 1
#3 bBusy6 <= #1.out 2
#4 bLB06_TILL <= #0
#5 HUS1_LB06_DRIFTLAGE <= #1.out 4
#6 HUS1_LB06_L1 <= #1.out 5
#7 HUS1_LB06_L2 <= #1.out 6
#8 HUS1_LB06_PV01_IT <= #1.out 7
#9 HUS1_LB06_GP11_MV <= #1.out 8
#10 HUS1_LB06_GP12_MV <= #1.out 9
#11 HUS1_LB06_GF41_MV <= #1.out 10
#12 HUS1_LB06_GF42_MV <= #1.out 11
#13 HUS1_LB06_GP61_MV <= #1.out 12
#14 HUS1_LB06_GP61_GV <= #1.out 13
#15 HUS1_LB06_GP62_MV <= #1.out 14
#16 HUS1_LB06_GP62_GV <= #1.out 15
#17 HUS1_LB06_TF01_R <= #1.out 16
#18 HUS1_LB06_FF01_R <= #1.out 17
#19 HUS1_LB06_SFP_MV <= #1.out 18
#20 HUS1_LB06_GT11_MV <= #1.out 19
#21 HUS1_LB06_GT31_MV <= #1.out 21
#22 HUS1_LB06_GT81_MV <= #1.out 22
#23 HUS1_LB06_VVX01_VVX <= #1.out 23
#24 HUS1_LB06_SV21_R <= #1.out 24
#25 KOMFEL_DELAY:fbDelayedAlarmMinutes(_bLarm: #1.out 1, _iMinutes: HUS1_LB06_LC_FL)
#26 HUS1_LB06_LC <= #25.bDelayedAlarm
#27 INT_TO_REAL(LB06_MODBUS.stGOLD.InputRegs2.EA_temperature_RX)
#28 DIV(#27, 100)
#29 HUS1_LB06_GT41_MV <= #28
_END_CFC_
END_PROGRAM

(* POU SYSTEM/HUS2_AS01_MAIN, CFC *)
PROGRAM HUS2_AS01_MAIN
VAR
	fbHelg: fbDFH_HD;
	DFH_Aktiv: BOOL;
	HD_Aktiv: BOOL;


END_VAR
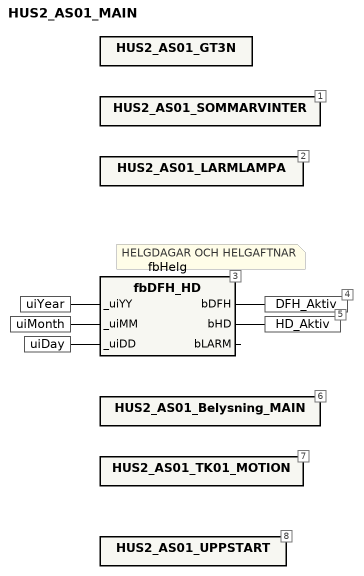
_CFC_ (* Continuous Function Chart, elements in execution order *)
(* HELGDAGAR OCH HELGAFTNAR *)
#0 HUS2_AS01_GT3N()
#1 HUS2_AS01_SOMMARVINTER()
#2 HUS2_AS01_LARMLAMPA()
#3 fbHelg:fbDFH_HD(_uiYY: uiYear, _uiMM: uiMonth, _uiDD: uiDay)
#4 DFH_Aktiv <= #3.bDFH
#5 HD_Aktiv <= #3.bHD
#6 HUS2_AS01_Belysning_MAIN()
#7 HUS2_AS01_TK01_MOTION()
#8 HUS2_AS01_UPPSTART()
_END_CFC_
(* the same logic as Structured Text *)
(* HELGDAGAR OCH HELGAFTNAR *)
HUS2_AS01_GT3N();
HUS2_AS01_SOMMARVINTER();
HUS2_AS01_LARMLAMPA();
fbHelg(_uiYY := uiYear, _uiMM := uiMonth, _uiDD := uiDay);
DFH_Aktiv := fbHelg.bDFH;
HD_Aktiv := fbHelg.bHD;
HUS2_AS01_Belysning_MAIN();
HUS2_AS01_TK01_MOTION();
HUS2_AS01_UPPSTART();
END_PROGRAM

(* POU xEgna Funktionsblock/fbDFH_HD, ST *)
FUNCTION_BLOCK fbDFH_HD

(*
Helgdagar och helgaftnar enligt: kalender.se
*)

VAR_INPUT
	_uiYY:				UINT;		(* Årtal i YY-format *)
	_uiMM:			UINT;		(*Månad i MM-format *)
	_uiDD:				UINT;		(*Dag i månaden i DD-format *)
END_VAR
VAR_OUTPUT
	bDFH:				BOOL;		(*	Helgafton/dag före helg*)
	bHD:				BOOL;		(* Helgdag/röd dag*)
	bLARM:			BOOL; 	(* Larmflagga, "slut" på kalender*)
END_VAR

VAR
	_rDatum:			DINT;		(*Aktuellt datum, YYMMDD*)
	AktuellDatumArray: 	ARRAY [1..22] OF DINT;
END_VAR

VAR CONSTANT

(*Datumarrays med helgdagar/-aftnar mellan år 2017-2037*)
	Array2017	:ARRAY [1..22] OF DINT :=		170105,	170413,	170415,	170430,	170603,	170623,	171103,	171224,	171231,	170101,	170106,	170414,	170416,	170417,	170501,	170525,	170604,	170606,	170624,	171104,	171225,	171226;
	Array2018	:ARRAY [1..22] OF DINT :=		180105,	180329,	180331,	180430,	180519,	180622,	181102,	181224,	181231,	180101,	180106,	180330,	180401,	180402,	180501,	180510,	180520,	180606,	180623,	181103,	181225,	181226;	
	Array2019	:ARRAY [1..22] OF DINT :=		190105,	190418,	190420,	190430,	190608,	190621,	191101,	191224,	191231,	190101,	190106,	190419,	190421,	190422,	190501,	190530,	190606,	190606,	190622,	191102,	191225,	191226;	
	Array2020	:ARRAY [1..22] OF DINT :=		200105,	200409,	200411,	200430,	200530,	200619,	201106,	201224,	201231,	200101,	200106,	200410,	200412,	200413,	200501,	200521,	200531,	200606,	200620,	201031,	201225,	201226;	
	Array2021	:ARRAY [1..22] OF DINT :=		210105,	210401,	210403,	210430,	210522,	210625,	211105,	211224,	211231,	210101,	210106,	210402,	210404,	210405,	210501,	210513,	210523,	210606,	210626,	211106,	211225,	211226;	
	Array2022	:ARRAY [1..22] OF DINT :=		220105,	220414,	220416,	220430,	220604,	220624,	221104,	221224,	221231,	220101,	220106,	220415,	220417,	220418,	220501,	220526,	220605,	220606,	220625,	221105,	221225,	221226;
	Array2023	:ARRAY [1..22] OF DINT :=		230105,	230406,	230408,	230430,	230527,	230623,	231103,	231224,	231231,	230101,	230106,	230407,	230409,	230410,	230501,	230518,	230528,	230606,	230624,	231104,	231225,	231226;	
	Array2024	:ARRAY [1..22] OF DINT :=		240105,	240328,	240330,	240430,	240518,	240621,	241101,	241224,	311231,	240101,	240106,	240329,	240331,	240401,	240501,	240509,	240519,	240606,	240622,	241102,	241225,	241226;	
	Array2025	:ARRAY [1..22] OF DINT :=		250105,	250417,	250419,	250430,	250607,	250620,	251031,	251224,	251231,	250101,	250106,	250418,	250420,	250421,	250501,	250529,	250606,	250606,	250621,	251101,	251225,	251226;	
	Array2026	:ARRAY [1..22] OF DINT :=		260105,	260402,	260404,	260430,	260523,	260619,	261106,	261224,	261231,	260101,	260106,	260403,	260405,	260406,	260501,	260515,	260524,	260606,	260620,	261031,	261225,	261226;	
	Array2027	:ARRAY [1..22] OF DINT :=		270105,	270325,	270327,	270430,	270515,	270625,	271105,	271224,	271231,	270101,	270106,	270326,	270328,	270329,	270501,	270506,	270516,	270606,	270626,	271106,	271225,	271226;	
	Array2028	:ARRAY [1..22] OF DINT :=		280105,	280413,	280415,	280430,	280603,	280623,	281103,	281224,	281231,	280101,	280106,	280414,	280416,	280417,	280501,	280525,	280604,	280606,	280624,	281104,	281225,	281226;
	Array2029	:ARRAY [1..22] OF DINT :=		290105,	290329,	290331,	290430,	290519,	290622,	291102,	291224,	291231,	290101,	290106,	290330,	290401,	290402,	290501,	290510,	290520,	290606,	290623,	291103,	291225,	291226;	
	Array2030	:ARRAY [1..22] OF DINT :=		300105,	300418,	300420,	300430,	300608,	300621,	301101,	301224,	301231,	300101,	300106,	300419,	300421,	300422,	300501,	300530,	300606,	300606,	300622,	301102,	301225,	301226;	
	Array2031	:ARRAY [1..22] OF DINT :=		310105,	310410,	310412,	310430,	310531,	310620,	311031,	311224,	311231,	310101,	310106,	310411,	310413,	310414,	310504,	310522,	310601,	310606,	310621,	311101,	311225,	311226;	
	Array2032	:ARRAY [1..22] OF DINT :=		320105,	320325,	320327,	320430,	320515,	320625,	321105,	321224,	321231,	320101,	320106,	320326,	320328,	320329,	320501,	320506,	320516,	320606,	320626,	321106,	321225,	321226;	
	Array2033	:ARRAY [1..22] OF DINT :=		330105,	330414,	330416,	330430,	330604,	330624,	331104,	331224,	331231,	330101,	330106,	330415,	330417,	330418,	330501,	330526,	330605,	330606,	330625,	331105,	331225,	331226;	
	Array2034	:ARRAY [1..22] OF DINT :=		340105,	340406,	340408,	340430,	340527,	340623,	341103,	341224,	341231,	340101,	340106,	340407,	340409,	340410,	340501,	340518,	340528,	340606,	340624,	341104,	341225,	341226;	
	Array2035	:ARRAY [1..22] OF DINT :=		350105,	350322,	350324,	350430,	350512,	350622,	351102,	351224,	351231,	350101,	350106,	350323,	350325,	350326,	350501,	350503,	350513,	350606,	350623,	351103,	351225,	351226;	
	Array2036	:ARRAY [1..22] OF DINT :=		360105,	360410,	360412,	360430,	360531,	360620,	361031,	361224,	361231,	360101,	360106,	360411,	360413,	360414,	360501,	360522,	360601,	360606,	360621,	361101,	361225,	361226;	
	Array2037	:ARRAY [1..22] OF DINT :=		370105,	370402,	370404,	370430,	370523,	370619,	371106,	371224,	371231,	370101,	370106,	370403,	370405,	370406,	370501,	370514,	370524,	370606,	370620,	371031,	371225,	371226;	

(*
Arrayförklaring:
Aftnar:
	ArrayXXXX[1] = 	Trettondagsafton	
	ArrayXXXX[2] = 	Skartorsdag	
	ArrayXXXX[3] = 	Paskafton	
	ArrayXXXX[4] = 	Valborgsmassoafton	
	ArrayXXXX[5] = 	Pingstafton	
	ArrayXXXX[6] = 	Midsommarafton	
	ArrayXXXX[7] = 	AllaHelgonsAfton	
	ArrayXXXX[8] = 	Julafton	
	ArrayXXXX[9] = 	Nyarsafton	
Dagar:
	ArrayXXXX[10] = 	Nyarsdagen	
	ArrayXXXX[11] = 	TrettondagJul	
	ArrayXXXX[12] = 	Langfredag	
	ArrayXXXX[13] = 	Paskdagen	
	ArrayXXXX[14] = 	AnnandagPask	
	ArrayXXXX[15] = 	ForstaMaj	
	ArrayXXXX[16] = 	KristiHimmelsfard	
	ArrayXXXX[17] = 	Pingstdagen	
	ArrayXXXX[18] = 	Nationaldagen	
	ArrayXXXX[19] = 	Midsommardagen	
	ArrayXXXX[20] = 	AllaHelgonsDag	
	ArrayXXXX[21] = 	Juldagen	
	ArrayXXXX[22] = 	AnnandagJul	

*)
END_VAR
(* Beräkna aktuellt datum i YYMMDD-format *)
_rDatum:=(_uiYY-2000)*10000 + (_uiMM*100)+_uiDD;

